	TCOM_STATE.TCOM_STATE_OP:
		// Check mapping of state:
		_bIsStateMapped := (F_GetMappingStatus(ADR(nRawState), SIZEOF(nRawState)) <> EPlcMappingStatus.MS_Unmapped);
		// Check mapping of overridden IO:
		_bIsOverriddenMapped := (F_GetMappingStatus(ADR(bRawOverridden), SIZEOF(bRawOverridden)) <> EPlcMappingStatus.MS_Unmapped);

END_CASE
END_METHOD

END_FUNCTION_BLOCK

// POUs/Local/Objects/5P/FB_BACnet_AO_Raw5P
// Analog Output Object
// - Raw communication
// - 5 Priorities
FUNCTION_BLOCK FB_BACnet_AO_Raw5P EXTENDS FB_BACnet_AO_Raw
VAR_INPUT
	bEnSfty					: BOOL;
	fValSfty				: REAL;
	bEnCrit					: BOOL;
	fValCrit				: REAL;
	bEnManLoc				: BOOL;
	fValManLoc				: REAL;
END_VAR
VAR_INPUT CONSTANT PERSISTENT
	{region 'Operational Parameters'}
		{attribute 'parameterCategory':='Manual'}
		bEnManualRm : BOOL;
		{attribute 'parameterCategory':='Manual'}
		fValManualRm : REAL;
	{endregion}
END_VAR
VAR_OUTPUT
	nActivePrio				: UDINT;			// Indicates the currently active priority of the priority array
END_VAR

SUPER^();

METHOD PROTECTED OnObjectStateChanged
SUPER^.OnObjectStateChanged();

CASE (tState) OF
	TCOM_STATE.TCOM_STATE_PREOP:
		// SyncHandler:
		RequestSyncHandlers(1, 4);
		
	TCOM_STATE.TCOM_STATE_SAFEOP:
		SyncProperty(E_BACnetPropIdentifier.PropCurrentlyActivePriority, SIZEOF(nActivePrio), ADR(nActivePrio), 0, eSync_FromSupplement, TRUE);

		SyncPropertyPvPrio(E_BACnetPropIdentifier.PropPresentValue, SIZEOF(fValSfty), ADR(fValSfty), ADR(bEnSfty), BACnet_Param.nPrio_LifeSafety, 0, eFullSync_InitPLC, TRUE);
		SyncPropertyPvPrio(E_BACnetPropIdentifier.PropPresentValue, SIZEOF(fValCrit), ADR(fValCrit), ADR(bEnCrit), BACnet_Param.nPrio_Critical, 0, eFullSync_InitPLC, TRUE);
		SyncPropertyPvPrio(E_BACnetPropIdentifier.PropPresentValue, SIZEOF(fValManLoc), ADR(fValManLoc), ADR(bEnManLoc), BACnet_Param.nPrio_ManLocal, 0, eFullSync_InitPLC, TRUE);
		SyncPropertyPvPrio(E_BACnetPropIdentifier.PropPresentValue, SIZEOF(fValManualRm), ADR(fValManualRm), ADR(bEnManualRm), BACnet_Param.nPrio_ManRemote, 0, eFullSync_InitPLC, TRUE);
		
	TCOM_STATE.TCOM_STATE_OP:
		;
		
END_CASE
END_METHOD

PROPERTY ActivePrio : UDINT
GET
ActivePrio := nActivePrio;
END_GET
END_PROPERTY

PROPERTY EnManualRm : BOOL
GET
EnManualRm := bEnManualRm;
END_GET
SET
bEnManualRm := EnManualRm;
END_SET
END_PROPERTY

PROPERTY ValManualRm : REAL
GET
ValManualRm := fValManualRm;
END_GET
SET
fValManualRm := ValManualRm;
END_SET
END_PROPERTY

END_FUNCTION_BLOCK

// POUs/Local/Objects/FB_BACnet_AO_Raw
// Analog Output Object
// - Raw communication
// - 1 Priority
FUNCTION_BLOCK FB_BACnet_AO_Raw EXTENDS FB_BACnet_BaseAO
VAR_INPUT
	bRawOverridden				: BOOL;				// Raw overridden
END_VAR
VAR_OUTPUT
	nRawValue					: INT;				// Raw value
END_VAR

IF (bReady) THEN
	// Overridden IO:
	_bOverriddenValue := bRawOverridden;
END_IF

SUPER^();

METHOD PROTECTED OnObjectStateChanged
SUPER^.OnObjectStateChanged();

CASE (tState) OF
	TCOM_STATE.TCOM_STATE_PREOP:
		// SyncHandler:
		RequestSyncHandlers(1, 0);

	TCOM_STATE.TCOM_STATE_SAFEOP:
		SyncProperty(E_BACnetPropIdentifier.PropRawIoAnalogValueINT, SIZEOF(nRawValue), ADR(nRawValue), 0, eSync_FromSupplement, TRUE);
		
	TCOM_STATE.TCOM_STATE_OP:
		;

END_CASE
END_METHOD

END_FUNCTION_BLOCK

// POUs/Local/Objects/5P/FB_BACnet_AV_5P
// Analog Value Object
// - 5 Priorities
FUNCTION_BLOCK FB_BACnet_AV_5P EXTENDS FB_BACnet_AV
VAR_INPUT
	bEnSfty					: BOOL;
	fValSfty				: REAL;
	bEnCrit					: BOOL;
	fValCrit				: REAL;
	bEnManLoc				: BOOL;
	fValManLoc				: REAL;
END_VAR
VAR_INPUT CONSTANT PERSISTENT
	{region 'Operational Parameters'}
		{attribute 'parameterCategory':='Manual'}
		bEnManualRm : BOOL;
		{attribute 'parameterCategory':='Manual'}
		fValManualRm : REAL;
	{endregion}
END_VAR
VAR_OUTPUT
	nActivePrio				: UDINT;			// Indicates the currently active priority of the priority array
END_VAR

SUPER^();

METHOD PROTECTED OnObjectStateChanged
SUPER^.OnObjectStateChanged();

CASE (tState) OF
	TCOM_STATE.TCOM_STATE_PREOP:
		// SyncHandler:
		RequestSyncHandlers(1, 4);
		
	TCOM_STATE.TCOM_STATE_SAFEOP:
		SyncProperty(E_BACnetPropIdentifier.PropCurrentlyActivePriority, SIZEOF(nActivePrio), ADR(nActivePrio), 0, eSync_FromSupplement, TRUE);

		SyncPropertyPvPrio(E_BACnetPropIdentifier.PropPresentValue, SIZEOF(fValSfty), ADR(fValSfty), ADR(bEnSfty), BACnet_Param.nPrio_LifeSafety, 0, eFullSync_InitPLC, TRUE);
		SyncPropertyPvPrio(E_BACnetPropIdentifier.PropPresentValue, SIZEOF(fValCrit), ADR(fValCrit), ADR(bEnCrit), BACnet_Param.nPrio_Critical, 0, eFullSync_InitPLC, TRUE);
		SyncPropertyPvPrio(E_BACnetPropIdentifier.PropPresentValue, SIZEOF(fValManLoc), ADR(fValManLoc), ADR(bEnManLoc), BACnet_Param.nPrio_ManLocal, 0, eFullSync_InitPLC, TRUE);
		SyncPropertyPvPrio(E_BACnetPropIdentifier.PropPresentValue, SIZEOF(fValManualRm), ADR(fValManualRm), ADR(bEnManualRm), BACnet_Param.nPrio_ManRemote, 0, eFullSync_InitPLC, TRUE);
		
	TCOM_STATE.TCOM_STATE_OP:
		;
	
END_CASE
END_METHOD

PROPERTY ActivePrio : UDINT
GET
ActivePrio := nActivePrio;
END_GET
END_PROPERTY

PROPERTY EnManualRm : BOOL
GET
EnManualRm := bEnManualRm;
END_GET
SET
bEnManualRm := EnManualRm;
END_SET
END_PROPERTY

PROPERTY ValManualRm : REAL
GET
ValManualRm := fValManualRm;
END_GET
SET
fValManualRm := ValManualRm;
END_SET
END_PROPERTY

END_FUNCTION_BLOCK

// POUs/Local/Objects/FB_BACnet_AV
// Analog Value Object
// - 1 Priority
FUNCTION_BLOCK FB_BACnet_AV EXTENDS FB_BACnet_EventObject
VAR_INPUT
	bEnPgm			: BOOL;
	fValPgm			: REAL;
END_VAR
VAR_INPUT CONSTANT PERSISTENT
	{region 'Variable Parameters'}
		{attribute 'parameterCategory':='Value'}
		fRelinquishDefault : REAL;
		{attribute 'parameterCategory':='Value'}
		bEnOutOfService : BOOL;
		{attribute 'parameterCategory':='Value'}
		fCOVIncrement : REAL := 0.1;
		{attribute 'parameterCategory':='Value'}
		eUnit : E_BA_Unit := E_BA_Unit.eOther_NoUnits;
		
		{attribute 'parameterCategory':='EventConfig'}
		bLowLimitEnable : BOOL := FALSE;
		{attribute 'parameterCategory':='EventConfig'}
		fLowLimitValue : REAL;
		{attribute 'parameterCategory':='EventConfig'}
		bHighLimitEnable : BOOL := FALSE;
		{attribute 'parameterCategory':='EventConfig'}
		fHighLimitValue : REAL;
		{attribute 'parameterCategory':='EventConfig'}
		fDeadband : REAL := 0.0;
	{endregion}
END_VAR
VAR_OUTPUT
	fPresentValue	: REAL;
END_VAR

SUPER^();

METHOD PROTECTED OnObjectStateChanged
SUPER^.OnObjectStateChanged();

CASE (tState) OF
	TCOM_STATE.TCOM_STATE_PREOP:
		// SyncHandler:
		RequestSyncHandlers(0, 9);
		
		// DisableProperty(E_BACnetPropIdentifier.PropDeviceType);

	TCOM_STATE.TCOM_STATE_SAFEOP:
		SyncPropertyPvPrio(E_BACnetPropIdentifier.PropPresentValue, SIZEOF(fValPgm), ADR(fValPgm), ADR(bEnPgm), BACnet_Param.nPrio_Program, 0, eFullSync_InitPLC, TRUE);
		
		SyncProperty(E_BACnetPropIdentifier.PropPresentValue, SIZEOF(fPresentValue), ADR(fPresentValue), 0, eSync_FromSupplement, TRUE);
		
	TCOM_STATE.TCOM_STATE_OP:
		SyncProperty(E_BACnetPropIdentifier.PropUnits, SIZEOF(eUnit), ADR(eUnit), 0, eFullSync_InitPLC, FALSE);
		SyncPropertyIdx(E_BACnetPropIdentifier.PropLimitEnable, SIZEOF(BOOL), ADR(bHighLimitEnable), E_BACnet_LimitEnableBits.eHighLimit, 0, eFullSync_InitPLC, FALSE);	
		SyncPropertyIdx(E_BACnetPropIdentifier.PropLimitEnable, SIZEOF(BOOL), ADR(bLowLimitEnable), E_BACnet_LimitEnableBits.eLowLimit, 0, eFullSync_InitPLC, FALSE);
		SyncProperty(E_BACnetPropIdentifier.PropHighLimit, SIZEOF(fHighLimitValue), ADR(fHighLimitValue), 0, eFullSync_InitPLC, FALSE);
		SyncProperty(E_BACnetPropIdentifier.PropLowLimit, SIZEOF(fLowLimitValue), ADR(fLowLimitValue), 0, eFullSync_InitPLC, FALSE);
		SyncProperty(E_BACnetPropIdentifier.PropDeadband, SIZEOF(fDeadband), ADR(fDeadband), 0, eFullSync_InitPLC, FALSE);
		SyncProperty(E_BACnetPropIdentifier.PropRelinquishDefault, SIZEOF(fRelinquishDefault), ADR(fRelinquishDefault), 0, eFullSync_InitPLC, FALSE);
		SyncProperty(E_BACnetPropIdentifier.PropOutOfService, SIZEOF(bEnOutOfService), ADR(bEnOutOfService), 0, eFullSync_InitPLC, FALSE);
		SyncProperty(E_BACnetPropIdentifier.PropCovIncrement, SIZEOF(fCOVIncrement), ADR(fCOVIncrement), 0, eFullSync_InitPLC, FALSE);
END_CASE
END_METHOD

METHOD FB_init : BOOL
VAR_INPUT
	bInitRetains : BOOL; // if TRUE, the retain variables are initialized (warm start / cold start)
	bInCopyCode : BOOL;  // if TRUE, the instance afterwards gets moved into the copy code (online change)
END_VAR
eObjectType := E_BACnetObjType.ObjAnalogValue;
END_METHOD

END_FUNCTION_BLOCK

// POUs/Local/Objects/5P/FB_BACnet_BO_IO5P
// Binary Output Object
// - Terminal communication
// - 5 Priorities
FUNCTION_BLOCK FB_BACnet_BO_IO5P EXTENDS FB_BACnet_BO_IO
VAR_INPUT
	bEnSfty					: BOOL;
	bValSfty				: BOOL;
	bEnCrit					: BOOL;
	bValCrit				: BOOL;
	bEnManLoc				: BOOL;
	bValManLoc				: BOOL;
END_VAR
VAR_INPUT CONSTANT PERSISTENT
	{region 'Operational Parameters'}
		{attribute 'parameterCategory':='Manual'}
		bEnManualRm : BOOL;
		{attribute 'parameterCategory':='Manual'}
		bValManualRm : BOOL;
	{endregion}
END_VAR
VAR_OUTPUT
	nActivePrio				: UDINT;			// Indicates the currently active priority of the priority array
END_VAR

SUPER^();

METHOD PROTECTED OnObjectStateChanged
SUPER^.OnObjectStateChanged();

CASE (tState) OF
	TCOM_STATE.TCOM_STATE_PREOP:
		// SyncHandler:
		RequestSyncHandlers(1, 4);
		
	TCOM_STATE.TCOM_STATE_SAFEOP:
		SyncProperty(E_BACnetPropIdentifier.PropCurrentlyActivePriority, SIZEOF(nActivePrio), ADR(nActivePrio), 0, eSync_FromSupplement, TRUE);

		SyncPropertyPvPrio(E_BACnetPropIdentifier.PropPresentValue, SIZEOF(bValSfty), ADR(bValSfty), ADR(bEnSfty), BACnet_Param.nPrio_LifeSafety, 0, eFullSync_InitPLC, TRUE);
		SyncPropertyPvPrio(E_BACnetPropIdentifier.PropPresentValue, SIZEOF(bValCrit), ADR(bValCrit), ADR(bEnCrit), BACnet_Param.nPrio_Critical, 0, eFullSync_InitPLC, TRUE);
		SyncPropertyPvPrio(E_BACnetPropIdentifier.PropPresentValue, SIZEOF(bValManLoc), ADR(bValManLoc), ADR(bEnManLoc), BACnet_Param.nPrio_ManLocal, 0, eFullSync_InitPLC, TRUE);
		SyncPropertyPvPrio(E_BACnetPropIdentifier.PropPresentValue, SIZEOF(bValManualRm), ADR(bValManualRm), ADR(bEnManualRm), BACnet_Param.nPrio_ManRemote, 0, eFullSync_InitPLC, TRUE);
		
	TCOM_STATE.TCOM_STATE_OP:
		;
		
END_CASE
END_METHOD

PROPERTY ActivePrio : UDINT
GET
ActivePrio := nActivePrio;
END_GET
END_PROPERTY

PROPERTY EnManualRm : BOOL
GET
EnManualRm := bEnManualRm;
END_GET
SET
bEnManualRm := EnManualRm;
END_SET
END_PROPERTY

PROPERTY ValManualRm : BOOL
GET
ValManualRm := bValManualRm;
END_GET
SET
bValManualRm := ValManualRm;
END_SET
END_PROPERTY

END_FUNCTION_BLOCK

// POUs/Local/Objects/FB_BACnet_BO_IO
// Binary Output Object
// - Terminal communication
// - 1 Priority
FUNCTION_BLOCK FB_BACnet_BO_IO EXTENDS FB_BACnet_BaseBO
VAR_INPUT CONSTANT PERSISTENT
	{region 'Variable Parameters'}
		{attribute 'parameterCategory':='Config'}
		eFeedbackPolarity : E_BA_Polarity := E_BA_Polarity.eNormal;
		{attribute 'parameterCategory':='Config'}
		eOverriddenPolarity : E_BA_Polarity := E_BA_Polarity.eNormal;
	{endregion}
END_VAR
VAR
	{region 'Raw I/O'}
		bRawOverridden		AT %I*	: BOOL;				// Raw overridden (Optional)
		bRawValFeedback		AT %I*	: BOOL;				// Raw feedback Value (Optional)
		bRawValue			AT %Q*	: BOOL;				// Raw value
	{endregion}
	{region 'Hardware'}
		_bIsFeedbackMapped			: BOOL;				// Indication to mapped hardware for feedback value
		_bIsOverriddenMapped		: BOOL;				// Indication to mapped hardware for overridden IO value
	{endregion}
	{region 'Internal'}
		_bOverriddenValue			: BOOL;
	{endregion}
END_VAR
VAR_STAT 
	// (BETA) ... Following symbols should be made non-static / thread safe!
	{region 'Temporary'}
		{attribute 'hide'}
		_bEnFeedback				: BOOL;
	{endregion}
END_VAR

IF (bReady) THEN
	// Overridden IO Value:
	_bOverriddenValue := SEL(_bIsOverriddenMapped, FALSE, (bRawOverridden = (eOverriddenPolarity=E_BA_Polarity.eNormal)));
	
	// Feedback Value:
	_bEnFeedback := SEL(_bIsFeedbackMapped, FALSE, NOT _bOverriddenValue);
	_bFeedbackValue := SEL(_bEnFeedback, bPresentValue, (bRawValFeedback = (eFeedbackPolarity=E_BA_Polarity.eNormal)));
END_IF

SUPER^();

METHOD PROTECTED OnObjectStateChanged
SUPER^.OnObjectStateChanged();

CASE (tState) OF
	TCOM_STATE.TCOM_STATE_PREOP:
		// SyncHandler:
		RequestSyncHandlers(1, 1);

	TCOM_STATE.TCOM_STATE_SAFEOP:
		SyncProperty(E_BACnetPropIdentifier.PropRawIoBinaryValueBOOL, SIZEOF(bRawValue), ADR(bRawValue), 0, eSync_FromSupplement, TRUE);
		
	TCOM_STATE.TCOM_STATE_OP:
		SyncProperty(E_BACnetPropIdentifier.PropRawIoStateOverrideInverted, SIZEOF(_bOverriddenValue), ADR(_bOverriddenValue), 0, eSync_ToSupplement, FALSE);

		// Check mapping of feedback:
		_bIsFeedbackMapped := (F_GetMappingStatus(ADR(bRawValFeedback), SIZEOF(bRawValFeedback)) <> EPlcMappingStatus.MS_Unmapped);
		// Check mapping of overridden IO:
		_bIsOverriddenMapped := (F_GetMappingStatus(ADR(bRawOverridden), SIZEOF(bRawOverridden)) <> EPlcMappingStatus.MS_Unmapped);
		
END_CASE
END_METHOD

END_FUNCTION_BLOCK

// POUs/Local/Objects/5P/FB_BACnet_BO_Raw5P
// Binary Output Object
// - Raw communication
// - 5 Priorities
FUNCTION_BLOCK FB_BACnet_BO_Raw5P EXTENDS FB_BACnet_BO_Raw
VAR_INPUT
	bEnSfty					: BOOL;
	bValSfty				: BOOL;
	bEnCrit					: BOOL;
	bValCrit				: BOOL;
	bEnManLoc				: BOOL;
	bValManLoc				: BOOL;
END_VAR
VAR_INPUT CONSTANT PERSISTENT
	{region 'Operational Parameters'}
		{attribute 'parameterCategory':='Manual'}
		bEnManualRm : BOOL;
		{attribute 'parameterCategory':='Manual'}
		bValManualRm : BOOL;
	{endregion}
END_VAR
VAR_OUTPUT
	nActivePrio				: UDINT;			// Indicates the currently active priority of the priority array
END_VAR

SUPER^();

METHOD PROTECTED OnObjectStateChanged
SUPER^.OnObjectStateChanged();

CASE (tState) OF
	TCOM_STATE.TCOM_STATE_PREOP:
		// SyncHandler:
		RequestSyncHandlers(1, 4);
		
	TCOM_STATE.TCOM_STATE_SAFEOP:
		SyncProperty(E_BACnetPropIdentifier.PropCurrentlyActivePriority, SIZEOF(nActivePrio), ADR(nActivePrio), 0, eSync_FromSupplement, TRUE);

		SyncPropertyPvPrio(E_BACnetPropIdentifier.PropPresentValue, SIZEOF(bValSfty), ADR(bValSfty), ADR(bEnSfty), BACnet_Param.nPrio_LifeSafety, 0, eFullSync_InitPLC, TRUE);
		SyncPropertyPvPrio(E_BACnetPropIdentifier.PropPresentValue, SIZEOF(bValCrit), ADR(bValCrit), ADR(bEnCrit), BACnet_Param.nPrio_Critical, 0, eFullSync_InitPLC, TRUE);
		SyncPropertyPvPrio(E_BACnetPropIdentifier.PropPresentValue, SIZEOF(bValManLoc), ADR(bValManLoc), ADR(bEnManLoc), BACnet_Param.nPrio_ManLocal, 0, eFullSync_InitPLC, TRUE);
		SyncPropertyPvPrio(E_BACnetPropIdentifier.PropPresentValue, SIZEOF(bValManualRm), ADR(bValManualRm), ADR(bEnManualRm), BACnet_Param.nPrio_ManRemote, 0, eFullSync_InitPLC, TRUE);
		
	TCOM_STATE.TCOM_STATE_OP:
		;
		
END_CASE
END_METHOD

PROPERTY ActivePrio : UDINT
GET
ActivePrio := nActivePrio;
END_GET
END_PROPERTY

PROPERTY EnManualRm : BOOL
GET
EnManualRm := bEnManualRm;
END_GET
SET
bEnManualRm := EnManualRm;
END_SET
END_PROPERTY

PROPERTY ValManualRm : BOOL
GET
ValManualRm := bValManualRm;
END_GET
SET
bValManualRm := ValManualRm;
END_SET
END_PROPERTY

END_FUNCTION_BLOCK

// POUs/Local/Objects/FB_BACnet_BO_Raw
// Binary Output Object
// - Raw communication
// - 1 Priority
FUNCTION_BLOCK FB_BACnet_BO_Raw EXTENDS FB_BACnet_BaseBO
VAR_INPUT
	bRawOverridden				: BOOL;				// Raw overridden

	bEnFeedback					: BOOL;				// Enable of writing to Feedback Value (optional)
	bRawValFeedback				: BOOL;				// Raw feedback Value
END_VAR
VAR_OUTPUT
	bRawValue					: BOOL;				// Raw value
END_VAR

IF (bReady) THEN
	// Feedback Value:
	_bFeedbackValue := SEL(bEnFeedback, bPresentValue, bRawValFeedback);
END_IF

SUPER^();

METHOD PROTECTED OnObjectStateChanged
SUPER^.OnObjectStateChanged();

CASE (tState) OF
	TCOM_STATE.TCOM_STATE_PREOP:
		// SyncHandler:
		RequestSyncHandlers(1, 1);

	TCOM_STATE.TCOM_STATE_SAFEOP:
		SyncProperty(E_BACnetPropIdentifier.PropRawIoBinaryValueBOOL, SIZEOF(bRawValue), ADR(bRawValue), 0, eSync_FromSupplement, TRUE);
		
	TCOM_STATE.TCOM_STATE_OP:
		SyncProperty(E_BACnetPropIdentifier.PropRawIoStateOverrideInverted, SIZEOF(bRawOverridden), ADR(bRawOverridden), 0, eSync_ToSupplement, FALSE);

END_CASE
END_METHOD

END_FUNCTION_BLOCK

// POUs/Local/Objects/5P/FB_BACnet_BV_5P
// Binary Value Object
// - 5 Priorities
FUNCTION_BLOCK FB_BACnet_BV_5P EXTENDS FB_BACnet_BV
VAR_INPUT
	bEnSfty					: BOOL;
	bValSfty				: BOOL;
	bEnCrit					: BOOL;
	bValCrit				: BOOL;
	bEnManLoc				: BOOL;
	bValManLoc				: BOOL;
END_VAR
VAR_INPUT CONSTANT PERSISTENT
	{region 'Operational Parameters'}
		{attribute 'parameterCategory':='Manual'}
		bEnManualRm : BOOL;
		{attribute 'parameterCategory':='Manual'}
		bValManualRm : BOOL;
	{endregion}
END_VAR
VAR_OUTPUT
	nActivePrio				: UDINT;			// Indicates the currently active priority of the priority array
END_VAR

SUPER^();

METHOD PROTECTED OnObjectStateChanged
SUPER^.OnObjectStateChanged();

CASE (tState) OF
	TCOM_STATE.TCOM_STATE_PREOP:
		// SyncHandler:
		RequestSyncHandlers(1, 4);
		
	TCOM_STATE.TCOM_STATE_SAFEOP:
		SyncProperty(E_BACnetPropIdentifier.PropCurrentlyActivePriority, SIZEOF(nActivePrio), ADR(nActivePrio), 0, eSync_FromSupplement, TRUE);

		SyncPropertyPvPrio(E_BACnetPropIdentifier.PropPresentValue, SIZEOF(bValSfty), ADR(bValSfty), ADR(bEnSfty), BACnet_Param.nPrio_LifeSafety, 0, eFullSync_InitPLC, TRUE);
		SyncPropertyPvPrio(E_BACnetPropIdentifier.PropPresentValue, SIZEOF(bValCrit), ADR(bValCrit), ADR(bEnCrit), BACnet_Param.nPrio_Critical, 0, eFullSync_InitPLC, TRUE);
		SyncPropertyPvPrio(E_BACnetPropIdentifier.PropPresentValue, SIZEOF(bValManLoc), ADR(bValManLoc), ADR(bEnManLoc), BACnet_Param.nPrio_ManLocal, 0, eFullSync_InitPLC, TRUE);
		SyncPropertyPvPrio(E_BACnetPropIdentifier.PropPresentValue, SIZEOF(bValManualRm), ADR(bValManualRm), ADR(bEnManualRm), BACnet_Param.nPrio_ManRemote, 0, eFullSync_InitPLC, TRUE);
		
	TCOM_STATE.TCOM_STATE_OP:
		;
		
END_CASE
END_METHOD

PROPERTY ActivePrio : UDINT
GET
ActivePrio := nActivePrio;
END_GET
END_PROPERTY

PROPERTY EnManualRm : BOOL
GET
EnManualRm := bEnManualRm;
END_GET
SET
bEnManualRm := EnManualRm;
END_SET
END_PROPERTY

PROPERTY ValManualRm : BOOL
GET
ValManualRm := bValManualRm;
END_GET
SET
bValManualRm := ValManualRm;
END_SET
END_PROPERTY

END_FUNCTION_BLOCK

// POUs/Local/Objects/FB_BACnet_BV
// Binary Value Object
// - 1 Priority
FUNCTION_BLOCK FB_BACnet_BV EXTENDS FB_BACnet_EventObject
VAR_INPUT
	bEnPgm		: BOOL;
	bValPgm		: BOOL;
END_VAR
VAR_INPUT CONSTANT PERSISTENT
	{region 'Variable Parameters'}
		{attribute 'parameterCategory':='General'}
		{attribute 'parameterUnit':= 's'}
		nMinimumOffTime : UDINT;
		{attribute 'parameterCategory':='General'}
		{attribute 'parameterUnit':= 's'}
		nMinimumOnTime : UDINT;
		
		{attribute 'parameterCategory':='Value'}
		bRelinquishDefault : BOOL;
		{attribute 'parameterCategory':='Value'}
		bEnOutOfService : BOOL;
		{attribute 'parameterCategory':='Value'}
		{attribute 'TcEncoding':='UTF-8'}
		sInactiveText : T_BACnet_StateText;
		{attribute 'parameterCategory':='Value'}
		{attribute 'TcEncoding':='UTF-8'}
		sActiveText : T_BACnet_StateText;
		
		{attribute 'parameterCategory':='EventConfig'}
		bAlarmValue : BOOL := TRUE;
			 
		{attribute 'parameterCategory':='StateChange'}
		nChangeOfStateCount : UDINT;
		
		{attribute 'parameterCategory':='ActiveTime'}
		{attribute 'parameterUnit':= 's'}
		nElapsedActiveTime : UDINT;
	{endregion}
END_VAR
VAR_OUTPUT
	bPresentValue	: BOOL;
END_VAR
VAR
	{region 'Output-Properties'}
		{attribute 'parameterCategory':='StateChange'}
		stChangeOfStateTime : ST_BA_DateTime;
		{attribute 'parameterCategory':='StateChange'}
		stTimeOfStateCountReset : ST_BA_DateTime;
		
		{attribute 'parameterCategory':='ActiveTime'}
		stTimeOfActiveTimeReset : ST_BA_DateTime;
	{endregion}
END_VAR

SUPER^();

METHOD PROTECTED OnObjectStateChanged
SUPER^.OnObjectStateChanged();

CASE (tState) OF
	TCOM_STATE.TCOM_STATE_PREOP:
		// SyncHandler:
		RequestSyncHandlers(4, 10);
		
		// Properties:
		EnableProperty(E_BACnetPropIdentifier.PropDeviceType, FALSE);

		IF (BACnet_Param.bStateText_WriteProtect) THEN
			WriteProtectProperty(E_BACnetPropIdentifier.PropActiveText, TRUE);
			WriteProtectProperty(E_BACnetPropIdentifier.PropInactiveText, TRUE);
		END_IF
		
		// Ensure UTF-8 Encoding:
		F_BA_EnsureUTF8(ADR(sInactiveText), SIZEOF(sInactiveText));
		F_BA_EnsureUTF8(ADR(sActiveText), SIZEOF(sActiveText));

	TCOM_STATE.TCOM_STATE_SAFEOP:
		SyncPropertyPvPrio(E_BACnetPropIdentifier.PropPresentValue, SIZEOF(bValPgm), ADR(bValPgm), ADR(bEnPgm), BACnet_Param.nPrio_Program, 0, eFullSync_InitPLC, TRUE);
		
		SyncProperty(E_BACnetPropIdentifier.PropPresentValue, SIZEOF(bPresentValue), ADR(bPresentValue), 0, eSync_FromSupplement, TRUE);
		
	TCOM_STATE.TCOM_STATE_OP:
		SyncProperty(E_BACnetPropIdentifier.PropAlarmValue, SIZEOF(bAlarmValue), ADR(bAlarmValue), 0, eFullSync_InitPLC, FALSE);
		SyncProperty(E_BACnetPropIdentifier.PropOutOfService, SIZEOF(bEnOutOfService), ADR(bEnOutOfService), 0, eFullSync_InitPLC, FALSE);
		SyncProperty(E_BACnetPropIdentifier.PropMinimumOffTime, SIZEOF(nMinimumOffTime), ADR(nMinimumOffTime), 0, eFullSync_InitPLC, FALSE);	
		SyncProperty(E_BACnetPropIdentifier.PropMinimumOnTime, SIZEOF(nMinimumOnTime), ADR(nMinimumOnTime), 0, eFullSync_InitPLC, FALSE);	
		SyncProperty(E_BACnetPropIdentifier.PropRelinquishDefault, SIZEOF(bRelinquishDefault), ADR(bRelinquishDefault), 0, eFullSync_InitPLC, FALSE);	
		SyncProperty(E_BACnetPropIdentifier.PropActiveText, SIZEOF(sActiveText), ADR(sActiveText), 0, eFullSync_InitPLC, FALSE);	
		SyncProperty(E_BACnetPropIdentifier.PropInactiveText, SIZEOF(sInactiveText), ADR(sInactiveText), 0, eFullSync_InitPLC, FALSE);

		SyncProperty(E_BACnetPropIdentifier.PropChangeOfStateCount, SIZEOF(nChangeOfStateCount), ADR(nChangeOfStateCount), 0, eFullSync_InitPLC, FALSE);
		SyncProperty(E_BACnetPropIdentifier.PropChangeOfStateTime, SIZEOF(stChangeOfStateTime), ADR(stChangeOfStateTime), 0, eSync_FromSupplement, FALSE);
		SyncProperty(E_BACnetPropIdentifier.PropTimeOfStateCountReset, SIZEOF(stTimeOfStateCountReset), ADR(stTimeOfStateCountReset), 0, eSync_FromSupplement, FALSE);

		SyncProperty(E_BACnetPropIdentifier.PropElapsedActiveTime, SIZEOF(nElapsedActiveTime), ADR(nElapsedActiveTime), 0, eFullSync_InitPLC, FALSE);
		SyncProperty(E_BACnetPropIdentifier.PropTimeOfActiveTimeReset, SIZEOF(stTimeOfActiveTimeReset), ADR(stTimeOfActiveTimeReset), 0, eSync_FromSupplement, FALSE);
		
END_CASE
END_METHOD

METHOD FB_init : BOOL
VAR_INPUT
	bInitRetains : BOOL; // if TRUE, the retain variables are initialized (warm start / cold start)
	bInCopyCode : BOOL;  // if TRUE, the instance afterwards gets moved into the copy code (online change)
END_VAR
eObjectType := E_BACnetObjType.ObjBinaryValue;
END_METHOD

END_FUNCTION_BLOCK

// POUs/Local/Objects/5P/FB_BACnet_MO_IO5P
// Multistate Output Object
// - Terminal communication
// - 5 Priorities
FUNCTION_BLOCK FB_BACnet_MO_IO5P EXTENDS FB_BACnet_MO_IO
VAR_INPUT
	bEnSfty					: BOOL;
	nValSfty				: UDINT		:= 1;
	bEnCrit					: BOOL;
	nValCrit				: UDINT		:= 1;
	bEnManLoc				: BOOL;
	nValManLoc				: UDINT		:= 1;
END_VAR
VAR_INPUT CONSTANT PERSISTENT
	{region 'Operational Parameters'}
		{attribute 'parameterCategory':='Manual'}
		bEnManualRm : BOOL;
		{attribute 'parameterCategory':='Manual'}
		nValManualRm : UDINT := 1;
	{endregion}
END_VAR
VAR_OUTPUT
	nActivePrio				: UDINT;					// Indicates the currently active priority of the priority array
END_VAR

SUPER^();

METHOD PROTECTED OnObjectStateChanged
SUPER^.OnObjectStateChanged();

CASE (tState) OF
	TCOM_STATE.TCOM_STATE_PREOP:
		// SyncHandler:
		RequestSyncHandlers(1, 4);
		
	TCOM_STATE.TCOM_STATE_SAFEOP:
		SyncProperty(E_BACnetPropIdentifier.PropCurrentlyActivePriority, SIZEOF(nActivePrio), ADR(nActivePrio), 0, eSync_FromSupplement, TRUE);

		SyncPropertyPvPrio(E_BACnetPropIdentifier.PropPresentValue, SIZEOF(nValSfty), ADR(nValSfty), ADR(bEnSfty), BACnet_Param.nPrio_LifeSafety, 0, eFullSync_InitPLC, TRUE);
		SyncPropertyPvPrio(E_BACnetPropIdentifier.PropPresentValue, SIZEOF(nValCrit), ADR(nValCrit), ADR(bEnCrit), BACnet_Param.nPrio_Critical, 0, eFullSync_InitPLC, TRUE);
		SyncPropertyPvPrio(E_BACnetPropIdentifier.PropPresentValue, SIZEOF(nValManLoc), ADR(nValManLoc), ADR(bEnManLoc), BACnet_Param.nPrio_ManLocal, 0, eFullSync_InitPLC, TRUE);
		SyncPropertyPvPrio(E_BACnetPropIdentifier.PropPresentValue, SIZEOF(nValManualRm), ADR(nValManualRm), ADR(bEnManualRm), BACnet_Param.nPrio_ManRemote, 0, eFullSync_InitPLC, TRUE);
		
	TCOM_STATE.TCOM_STATE_OP:
		;
		
END_CASE
END_METHOD

PROPERTY ActivePrio : UDINT
GET
ActivePrio := nActivePrio;
END_GET
END_PROPERTY

PROPERTY EnManualRm : BOOL
GET
EnManualRm := bEnManualRm;
END_GET
SET
bEnManualRm := EnManualRm;
END_SET
END_PROPERTY

PROPERTY ValManualRm : UDINT
GET
ValManualRm := nValManualRm;
END_GET
SET
nValManualRm := ValManualRm;
END_SET
END_PROPERTY

END_FUNCTION_BLOCK

// POUs/Local/Objects/FB_BACnet_MO_IO
// Multistate Output Object
// - Terminal communication
// - 1 Priority
FUNCTION_BLOCK FB_BACnet_MO_IO EXTENDS FB_BACnet_BaseMO
VAR_INPUT CONSTANT PERSISTENT
	{region 'Variable Parameters'}
		{attribute 'parameterCategory':='Config'}
		eMappingMode : E_BA_ByteMappingMode := E_BA_ByteMappingMode.eIndex1N;
		{attribute 'parameterCategory':='Config'}
		eFeedbackMappingMode : E_BA_ByteMappingMode := E_BA_ByteMappingMode.eIndex1N;
	{endregion}
END_VAR
VAR
	{region 'Raw I/O'}
		bRawValFeedback		AT %I*	: ST_BA_Byte;		// Bus terminal feedback Value (Optional)
		bRawValue			AT %Q*	: ST_BA_Byte;		// Bus terminal value
	{endregion}
	{region 'Hardware'}
		_bIsFeedbackMapped			: BOOL;				// Indication to mapped hardware for feedback value
	{endregion}
	{region 'Internal'}
		nLastPresentValue			: UDINT;
	{endregion}
END_VAR

IF (bReady) THEN
	// Feedback Value:
	IF (_bIsFeedbackMapped) THEN
		F_BA_MapUDIFromRawByte(bRawValFeedback, _nFeedbackValue, eFeedbackMappingMode, nRelinquishDefault);
	ELSE
		_nFeedbackValue := nPresentValue;
	END_IF
	
	// Trigger change of value:
	IF (nPresentValue <> nLastPresentValue) THEN
		nLastPresentValue := nPresentValue;
		F_BA_MapUDIToRawByte(bRawValue, nPresentValue, eMappingMode, nRelinquishDefault);
	END_IF
ELSE
	nPresentValue := nRelinquishDefault;
	
	// Set last value to a different value compared to actual raw value (So a COV is triggered when current instance becomes ready):
	nLastPresentValue := (nLastPresentValue+1);
END_IF

SUPER^();

METHOD PROTECTED OnObjectStateChanged
SUPER^.OnObjectStateChanged();

CASE (tState) OF
	TCOM_STATE.TCOM_STATE_PREOP:
		;

	TCOM_STATE.TCOM_STATE_SAFEOP:
		;
		
	TCOM_STATE.TCOM_STATE_OP:
		// Check mapping of feedback:
		_bIsFeedbackMapped := (F_GetMappingStatus(ADR(bRawValFeedback), SIZEOF(bRawValFeedback)) <> EPlcMappingStatus.MS_Unmapped);
		
END_CASE
END_METHOD

END_FUNCTION_BLOCK

// POUs/Local/Objects/5P/FB_BACnet_MO_Raw5P
// Multistate Output Object
// - Raw communication
// - 5 Priorities
FUNCTION_BLOCK FB_BACnet_MO_Raw5P EXTENDS FB_BACnet_MO_Raw
VAR_INPUT
	bEnSfty					: BOOL;
	nValSfty				: UDINT		:= 1;
	bEnCrit					: BOOL;
	nValCrit				: UDINT		:= 1;
	bEnManLoc				: BOOL;
	nValManLoc				: UDINT		:= 1;
END_VAR
VAR_INPUT CONSTANT PERSISTENT
	{region 'Operational Parameters'}
		{attribute 'parameterCategory':='Manual'}
		bEnManualRm : BOOL;
		{attribute 'parameterCategory':='Manual'}
		nValManualRm : UDINT := 1;
	{endregion}
END_VAR
VAR_OUTPUT
	nActivePrio				: UDINT;					// Indicates the currently active priority of the priority array
END_VAR

SUPER^();

METHOD PROTECTED OnObjectStateChanged
SUPER^.OnObjectStateChanged();

CASE (tState) OF
	TCOM_STATE.TCOM_STATE_PREOP:
		// SyncHandler:
		RequestSyncHandlers(1, 4);
		
	TCOM_STATE.TCOM_STATE_SAFEOP:
		SyncProperty(E_BACnetPropIdentifier.PropCurrentlyActivePriority, SIZEOF(nActivePrio), ADR(nActivePrio), 0, eSync_FromSupplement, TRUE);

		SyncPropertyPvPrio(E_BACnetPropIdentifier.PropPresentValue, SIZEOF(nValSfty), ADR(nValSfty), ADR(bEnSfty), BACnet_Param.nPrio_LifeSafety, 0, eFullSync_InitPLC, TRUE);
		SyncPropertyPvPrio(E_BACnetPropIdentifier.PropPresentValue, SIZEOF(nValCrit), ADR(nValCrit), ADR(bEnCrit), BACnet_Param.nPrio_Critical, 0, eFullSync_InitPLC, TRUE);
		SyncPropertyPvPrio(E_BACnetPropIdentifier.PropPresentValue, SIZEOF(nValManLoc), ADR(nValManLoc), ADR(bEnManLoc), BACnet_Param.nPrio_ManLocal, 0, eFullSync_InitPLC, TRUE);
		SyncPropertyPvPrio(E_BACnetPropIdentifier.PropPresentValue, SIZEOF(nValManualRm), ADR(nValManualRm), ADR(bEnManualRm), BACnet_Param.nPrio_ManRemote, 0, eFullSync_InitPLC, TRUE);
		
	TCOM_STATE.TCOM_STATE_OP:
		;
		
END_CASE
END_METHOD

PROPERTY ActivePrio : UDINT
GET
ActivePrio := nActivePrio;
END_GET
END_PROPERTY

PROPERTY EnManualRm : BOOL
GET
EnManualRm := bEnManualRm;
END_GET
SET
bEnManualRm := EnManualRm;
END_SET
END_PROPERTY

PROPERTY ValManualRm : UDINT
GET
ValManualRm := nValManualRm;
END_GET
SET
nValManualRm := ValManualRm;
END_SET
END_PROPERTY

END_FUNCTION_BLOCK

// POUs/Local/Objects/FB_BACnet_MO_Raw
// Multistate Output Object
// - Raw communication
// - 1 Priority
FUNCTION_BLOCK FB_BACnet_MO_Raw EXTENDS FB_BACnet_BaseMO
VAR_INPUT
	bEnFeedback					: BOOL;				// Enable of writing to Feedback Value (optional)
	nRawValFeedback				: UDINT;			// Raw feedback Value
END_VAR
VAR_OUTPUT
	nRawValue					: UDINT;			// Raw value
END_VAR

IF (bReady) THEN
	// Feedback Value:
	_nFeedbackValue := MAX(1, SEL(bEnFeedback, nPresentValue, nRawValFeedback));
	
	// Raw-IO Value:
	nRawValue := nPresentValue;
END_IF

SUPER^();

END_FUNCTION_BLOCK

// POUs/Local/Objects/5P/FB_BACnet_MV_5P
// Multistate Value Object
// - 5 Priorities
FUNCTION_BLOCK FB_BACnet_MV_5P EXTENDS FB_BACnet_MV
VAR_INPUT
	bEnSfty					: BOOL;
	nValSfty				: UDINT		:= 1;
	bEnCrit					: BOOL;
	nValCrit				: UDINT		:= 1;
	bEnManLoc				: BOOL;
	nValManLoc				: UDINT		:= 1;
END_VAR
VAR_INPUT CONSTANT PERSISTENT
	{region 'Operational Parameters'}
		{attribute 'parameterCategory':='Manual'}
		bEnManualRm : BOOL;
		{attribute 'parameterCategory':='Manual'}
		nValManualRm : UDINT := 1;
	{endregion}
END_VAR
VAR_OUTPUT
	nActivePrio				: UDINT;			// Indicates the currently active priority of the priority array
END_VAR

SUPER^();

METHOD PROTECTED OnObjectStateChanged
SUPER^.OnObjectStateChanged();

CASE (tState) OF
	TCOM_STATE.TCOM_STATE_PREOP:
		// SyncHandler:
		RequestSyncHandlers(1, 4);
		
	TCOM_STATE.TCOM_STATE_SAFEOP:
		SyncProperty(E_BACnetPropIdentifier.PropCurrentlyActivePriority, SIZEOF(nActivePrio), ADR(nActivePrio), 0, eSync_FromSupplement, TRUE);

		SyncPropertyPvPrio(E_BACnetPropIdentifier.PropPresentValue, SIZEOF(nValSfty), ADR(nValSfty), ADR(bEnSfty), BACnet_Param.nPrio_LifeSafety, 0, eFullSync_InitPLC, TRUE);
		SyncPropertyPvPrio(E_BACnetPropIdentifier.PropPresentValue, SIZEOF(nValCrit), ADR(nValCrit), ADR(bEnCrit), BACnet_Param.nPrio_Critical, 0, eFullSync_InitPLC, TRUE);
		SyncPropertyPvPrio(E_BACnetPropIdentifier.PropPresentValue, SIZEOF(nValManLoc), ADR(nValManLoc), ADR(bEnManLoc), BACnet_Param.nPrio_ManLocal, 0, eFullSync_InitPLC, TRUE);
		SyncPropertyPvPrio(E_BACnetPropIdentifier.PropPresentValue, SIZEOF(nValManualRm), ADR(nValManualRm), ADR(bEnManualRm), BACnet_Param.nPrio_ManRemote, 0, eFullSync_InitPLC, TRUE);
		
	TCOM_STATE.TCOM_STATE_OP:
		;
		
END_CASE
END_METHOD

PROPERTY ActivePrio : UDINT
GET
ActivePrio := nActivePrio;
END_GET
END_PROPERTY

PROPERTY EnManualRm : BOOL
GET
EnManualRm := bEnManualRm;
END_GET
SET
bEnManualRm := EnManualRm;
END_SET
END_PROPERTY

PROPERTY ValManualRm : UDINT
GET
ValManualRm := nValManualRm;
END_GET
SET
nValManualRm := ValManualRm;
END_SET
END_PROPERTY

END_FUNCTION_BLOCK

// POUs/Local/Objects/FB_BACnet_MV
// Multistate Value Object
// - 1 Priority
FUNCTION_BLOCK FB_BACnet_MV EXTENDS FB_BACnet_EventObject
VAR_INPUT
	bEnPgm					: BOOL;
	nValPgm					: UDINT		:= 1;
END_VAR
VAR_INPUT CONSTANT PERSISTENT
	{region 'Fixed Parameters'}
		{attribute 'parameterCategory':='Value'}
		{attribute 'TcEncoding':='UTF-8'}
		sStateText : ARRAY[1..BACnet_Param.nMultistate_StateCount] OF T_BACnet_StateText;
		
		{attribute 'parameterCategory':='EventConfig'}
		nAlarmValues : ARRAY[1..BACnet_Param.nMultistate_StateCount] OF UDINT;
		{attribute 'parameterCategory':='EventConfig'}
		nFaultValues : ARRAY[1..BACnet_Param.nMultistate_StateCount] OF UDINT;
	{endregion}
	{region 'Variable Parameters'}
		{attribute 'parameterCategory':='Value'}
		nRelinquishDefault : UDINT := 1;
		{attribute 'parameterCategory':='Value'}
		bEnOutOfService : BOOL;
	{endregion}
END_VAR
VAR_OUTPUT
	nPresentValue			: UDINT		:= 1;
END_VAR
VAR
	{region 'Output-Properties'}
		nStateCount			: UDINT;
	{endregion}
END_VAR

SUPER^();

METHOD PROTECTED OnObjectStateChanged
SUPER^.OnObjectStateChanged();

CASE (tState) OF
	TCOM_STATE.TCOM_STATE_PREOP:
		// SyncHandler:
		{warning disable C0196}
		nStateCount := F_BACnet_GetUsedStateText(sStateText);
		{warning restore C0196}
		
		RequestSyncHandlers(0, nStateCount);								// Handlers for "E_BACnetPropIdentifier.PropStateText"
		RequestSyncHandlers(0, F_BACnet_GetUsedUDINT(nAlarmValues));		// Handlers for "E_BACnetPropIdentifier.PropAlarmValues"
		RequestSyncHandlers(0, F_BACnet_GetUsedUDINT(nFaultValues));		// Handlers for "E_BACnetPropIdentifier.PropFaultValues"
		RequestSyncHandlers(1, 3);											// Handlers for other properties
		
		// Properties:
		EnableProperty(E_BACnetPropIdentifier.PropDeviceType, FALSE);
		
		WriteProtectProperty(E_BACnetPropIdentifier.PropNumberOfStates, TRUE);
		
		IF (BACnet_Param.bStateText_WriteProtect) THEN
			WriteProtectProperty(E_BACnetPropIdentifier.PropStateText, TRUE);
		END_IF
		
		// Ensure UTF-8 Encoding:
		F_BA_EnsureUTF8Array(ADR(sStateText), SIZEOF(sStateText[1]), TO_DINT(BACnet_Param.nMultistate_StateCount));
		
	TCOM_STATE.TCOM_STATE_SAFEOP:
		SyncPropertyPvPrio(E_BACnetPropIdentifier.PropPresentValue, SIZEOF(nValPgm), ADR(nValPgm), ADR(bEnPgm), BACnet_Param.nPrio_Program, 0, eFullSync_InitPLC, TRUE);
		
		SyncProperty(E_BACnetPropIdentifier.PropPresentValue, SIZEOF(nPresentValue), ADR(nPresentValue), 0, eSync_FromSupplement, TRUE);
		
	TCOM_STATE.TCOM_STATE_OP:
		// Init number of used states:
		SetNumberOfStates(nStateCount);
		
		SyncProperty(E_BACnetPropIdentifier.PropRelinquishDefault, SIZEOF(nRelinquishDefault), ADR(nRelinquishDefault), 0, eFullSync_InitPLC, FALSE);
		SyncProperty(E_BACnetPropIdentifier.PropOutOfService, SIZEOF(bEnOutOfService), ADR(bEnOutOfService), 0, eFullSync_InitPLC, FALSE);
		SyncPropertyList(E_BACnetPropIdentifier.PropStateText, ADR(sStateText), SIZEOF(T_BACnet_StateText), nStateCount, eFullSync_InitPLC, FALSE);
		SyncPropertyList(E_BACnetPropIdentifier.PropAlarmValues, ADR(nAlarmValues), SIZEOF(UDINT), nStateCount, eFullSync_InitPLC, TRUE);
		SyncPropertyList(E_BACnetPropIdentifier.PropFaultValues, ADR(nFaultValues), SIZEOF(UDINT), nStateCount, eFullSync_InitPLC, TRUE);
		
END_CASE
END_METHOD

METHOD FB_init : BOOL
VAR_INPUT
	bInitRetains : BOOL; // if TRUE, the retain variables are initialized (warm start / cold start)
	bInCopyCode : BOOL;  // if TRUE, the instance afterwards gets moved into the copy code (online change)
END_VAR
eObjectType := E_BACnetObjType.ObjMultistateValue;
END_METHOD

PROPERTY StateCount : UDINT
GET
StateCount := nStateCount;
END_GET
END_PROPERTY

END_FUNCTION_BLOCK

// POUs/Local/Objects/FB_BACnet_Acc
// Accumulator Object
FUNCTION_BLOCK FB_BACnet_Acc EXTENDS FB_BACnet_EventObject
VAR_OUTPUT
	nPresentValue			: UDINT;
END_VAR

SUPER^();

METHOD PROTECTED OnObjectStateChanged
SUPER^.OnObjectStateChanged();

CASE (tState) OF
	TCOM_STATE.TCOM_STATE_PREOP:
		// SyncHandler:
		RequestSyncHandlers(1, 0);
		
	TCOM_STATE.TCOM_STATE_SAFEOP:
		SyncProperty(E_BACnetPropIdentifier.PropPresentValue, SIZEOF(nPresentValue), ADR(nPresentValue), 0, eSync_FromSupplement, TRUE);
	
	TCOM_STATE.TCOM_STATE_OP:
		;
		
END_CASE
END_METHOD

METHOD FB_init : BOOL
VAR_INPUT
	bInitRetains : BOOL; // if TRUE, the retain variables are initialized (warm start / cold start)
	bInCopyCode : BOOL;  // if TRUE, the instance afterwards gets moved into the copy code (online change)
END_VAR
eObjectType := E_BACnetObjType.ObjAccumulator;
END_METHOD

END_FUNCTION_BLOCK

// POUs/Local/Objects/FB_BACnet_AI
// Analog Input Object
// - process value
FUNCTION_BLOCK FB_BACnet_AI EXTENDS FB_BACnet_BaseAI
VAR_INPUT
	fVal						: REAL;				// Process value
END_VAR

IF bReady THEN
	IF NOT bEnOutOfService THEN
		fPresentValue := fVal;
	END_IF
ELSE
	fPresentValue := 0;
END_IF

SUPER^();

METHOD PROTECTED OnObjectStateChanged
CASE (tState) OF
	TCOM_STATE.TCOM_STATE_PREOP:
		// SyncHandler:
		RequestSyncHandlers(0, 1);
		
		// Properties:
		EnableProperty(E_BACnetPropIdentifier.PropResolution, FALSE);
		EnableProperty(E_BACnetPropIdentifier.PropScaleOffset, FALSE);

	TCOM_STATE.TCOM_STATE_SAFEOP:
		SyncProperty(E_BACnetPropIdentifier.PropPresentValue, SIZEOF(fPresentValue), ADR(fPresentValue), 0, eFullSync_InitPLC, TRUE);
		
	TCOM_STATE.TCOM_STATE_OP:
		;

END_CASE

SUPER^.OnObjectStateChanged();
END_METHOD

END_FUNCTION_BLOCK

// POUs/Local/Objects/FB_BACnet_AI_IO
// Analog Input Object
// - Terminal communication
FUNCTION_BLOCK FB_BACnet_AI_IO EXTENDS FB_BACnet_BaseAI
VAR_INPUT CONSTANT PERSISTENT	
	{region 'Variable Parameters'}
		{attribute 'parameterCategory':='Hardware'}
		fResolution : REAL := 0.1;
		{attribute 'parameterCategory':='Hardware'}
		fScaleOffset : REAL := 0;
	{endregion}
END_VAR
VAR
	{region 'Raw I/O'}
		nRawState			AT %I*	: USINT;			// Bus terminal state
		nRawValue			AT %I*	: INT;				// Bus terminal value
	{endregion}
END_VAR

SUPER^();

METHOD PROTECTED OnObjectStateChanged
CASE (tState) OF
	TCOM_STATE.TCOM_STATE_PREOP:
		// SyncHandler:
		RequestSyncHandlers(1, 4);

	TCOM_STATE.TCOM_STATE_SAFEOP:
		SyncProperty(E_BACnetPropIdentifier.PropPresentValue, SIZEOF(fPresentValue), ADR(fPresentValue), 0, eSync_FromSupplement, TRUE);
		
		SyncProperty(E_BACnetPropIdentifier.PropRawIoStateUSINT, SIZEOF(nRawState), ADR(nRawState), 0, eSync_ToSupplement, TRUE);
		SyncProperty(E_BACnetPropIdentifier.PropRawIoAnalogValueINT, SIZEOF(nRawValue), ADR(nRawValue), 0, eSync_ToSupplement, TRUE);
		
	TCOM_STATE.TCOM_STATE_OP:
		SyncProperty(E_BACnetPropIdentifier.PropResolution, SIZEOF(fResolution), ADR(fResolution), 0, eFullSync_InitPLC, FALSE);
		SyncProperty(E_BACnetPropIdentifier.PropScaleOffset, SIZEOF(fScaleOffset), ADR(fScaleOffset), 0, eFullSync_InitPLC, FALSE);

END_CASE

SUPER^.OnObjectStateChanged();
END_METHOD

END_FUNCTION_BLOCK

// POUs/Local/Objects/FB_BACnet_AI_Raw
// Analog Input Object
// - Raw communication
FUNCTION_BLOCK FB_BACnet_AI_Raw EXTENDS FB_BACnet_BaseAI
VAR_INPUT
	nRawState					: USINT;			// Raw state
													// - Underrange:	0x01
													// - Overrange:		0x02
													// - Error:			0x04
	nRawValue					: INT;				// Raw value
END_VAR
VAR_INPUT CONSTANT PERSISTENT
	{region 'Variable Parameters'}
		{attribute 'parameterCategory':='Hardware'}
		fResolution : REAL := 0.1;
		{attribute 'parameterCategory':='Hardware'}
		fScaleOffset : REAL := 0
	{endregion};
END_VAR

SUPER^();

METHOD PROTECTED OnObjectStateChanged
CASE (tState) OF
	TCOM_STATE.TCOM_STATE_PREOP:
		// SyncHandler:
		RequestSyncHandlers(1, 4);

	TCOM_STATE.TCOM_STATE_SAFEOP:
		SyncProperty(E_BACnetPropIdentifier.PropPresentValue, SIZEOF(fPresentValue), ADR(fPresentValue), 0, eSync_FromSupplement, TRUE);
		
		SyncProperty(E_BACnetPropIdentifier.PropRawIoStateUSINT, SIZEOF(nRawState), ADR(nRawState), 0, eSync_ToSupplement, TRUE);
		SyncProperty(E_BACnetPropIdentifier.PropRawIoAnalogValueINT, SIZEOF(nRawValue), ADR(nRawValue), 0, eSync_ToSupplement, TRUE);
		
	TCOM_STATE.TCOM_STATE_OP:
		SyncProperty(E_BACnetPropIdentifier.PropResolution, SIZEOF(fResolution), ADR(fResolution), 0, eFullSync_InitPLC, FALSE);
		SyncProperty(E_BACnetPropIdentifier.PropScaleOffset, SIZEOF(fScaleOffset), ADR(fScaleOffset), 0, eFullSync_InitPLC, FALSE);

END_CASE


SUPER^.OnObjectStateChanged();
END_METHOD

END_FUNCTION_BLOCK

// POUs/Local/Objects/FB_BACnet_AV_Disp
// Analog Setpoint Object for Operation
// - Used to display a value
FUNCTION_BLOCK FB_BACnet_AV_Disp EXTENDS FB_BACnet_Object
VAR_INPUT
	fVal			: REAL;
END_VAR
VAR_INPUT CONSTANT PERSISTENT
	{region 'Variable Parameters'}
		{attribute 'parameterCategory':='Value'}
		fCOVIncrement : REAL := 0.1;
		{attribute 'parameterCategory':='Value'}
		eUnit : E_BA_Unit := E_BA_Unit.eOther_NoUnits;
	{endregion}
END_VAR
VAR_OUTPUT
	fPresentValue	: REAL;
END_VAR

IF bReady THEN
	fPresentValue := fVal;
ELSE
	fPresentValue := 0;
END_IF

SUPER^();

METHOD PROTECTED OnObjectStateChanged
SUPER^.OnObjectStateChanged();

CASE (tState) OF
	TCOM_STATE.TCOM_STATE_PREOP:
		// SyncHandler:
		RequestSyncHandlers(0, 3);
		
		// Properties:
		// EnableProperty(E_BACnetPropIdentifier.PropDeviceType, FALSE);
		EnableProperty(E_BACnetPropIdentifier.PropNotificationClass, FALSE);
		EnableProperty(E_BACnetPropIdentifier.PropNotifyType, FALSE);
		EnableProperty(E_BACnetPropIdentifier.PropEventEnable, FALSE);
		EnableProperty(E_BACnetPropIdentifier.PropEventTimeStamps, FALSE);
		EnableProperty(E_BACnetPropIdentifier.PropEventMessageTexts, FALSE);
		EnableProperty(E_BACnetPropIdentifier.PropEventMessageTextsConfig, FALSE);
		EnableProperty(E_BACnetPropIdentifier.PropTimeDelay, FALSE);
		EnableProperty(E_BACnetPropIdentifier.PropStatusFlags, FALSE);
		EnableProperty(E_BACnetPropIdentifier.PropAckedTransitions, FALSE);
		EnableProperty(E_BACnetPropIdentifier.PropReliability, FALSE);
		EnableProperty(E_BACnetPropIdentifier.PropEventState, FALSE);
		EnableProperty(E_BACnetPropIdentifier.PropEventDetectionEnable, FALSE);
		EnableProperty(E_BACnetPropIdentifier.PropEventAlgorithmInhibit, FALSE);
		EnableProperty(E_BACnetPropIdentifier.PropTimeDelayNormal, FALSE);
		EnableProperty(E_BACnetPropIdentifier.PropReliabilityEvaluationInhibit, FALSE);
		EnableProperty(E_BACnetPropIdentifier.PropLimitEnable, FALSE);
		EnableProperty(E_BACnetPropIdentifier.PropHighLimit, FALSE);
		EnableProperty(E_BACnetPropIdentifier.PropLowLimit, FALSE);
		EnableProperty(E_BACnetPropIdentifier.PropDeadband, FALSE);
		EnableProperty(E_BACnetPropIdentifier.PropRelinquishDefault, FALSE);
		EnableProperty(E_BACnetPropIdentifier.PropPriorityArray, FALSE);
		EnableProperty(E_BACnetPropIdentifier.PropOutOfService, FALSE);
		EnableProperty(E_BACnetPropIdentifier.PropCurrentlyActivePriority, FALSE);
		
		WriteProtectProperty(E_BACnetPropIdentifier.PropPresentValue, TRUE);
		
	TCOM_STATE.TCOM_STATE_SAFEOP:
		SyncProperty(E_BACnetPropIdentifier.PropPresentValue, SIZEOF(fVal), ADR(fVal), 0, eSync_ToSupplement, TRUE);
		
	TCOM_STATE.TCOM_STATE_OP:
		SyncProperty(E_BACnetPropIdentifier.PropUnits, SIZEOF(eUnit), ADR(eUnit), 0, eFullSync_InitPLC, FALSE);
		SyncProperty(E_BACnetPropIdentifier.PropCovIncrement, SIZEOF(fCOVIncrement), ADR(fCOVIncrement), 0, eFullSync_InitPLC, FALSE);
END_CASE
END_METHOD

METHOD FB_init : BOOL
VAR_INPUT
	bInitRetains : BOOL; // if TRUE, the retain variables are initialized (warm start / cold start)
	bInCopyCode : BOOL;  // if TRUE, the instance afterwards gets moved into the copy code (online change)
END_VAR
eObjectType := E_BACnetObjType.ObjAnalogValue;
END_METHOD

END_FUNCTION_BLOCK

// POUs/Local/Objects/FB_BACnet_AV_Setp
// Analog Setpoint Object for Operation
// - Used to define a setpoint by user
FUNCTION_BLOCK FB_BACnet_AV_Setp EXTENDS FB_BACnet_Object
VAR_INPUT CONSTANT PERSISTENT
	{region 'Variable Parameters'}
		{attribute 'parameterCategory':='Value'}
		fCOVIncrement : REAL := 0.1;
		{attribute 'parameterCategory':='Value'}
		eUnit : E_BA_Unit := E_BA_Unit.eOther_NoUnits;
	{endregion}
	{region 'Operational Parameters'}
		{attribute 'parameterCategory':='Value'}
		fValue : REAL;
	{endregion}
END_VAR
VAR_OUTPUT
	fPresentValue	: REAL;
END_VAR

IF bReady THEN
	fPresentValue := fValue;
ELSE
	fPresentValue := 0;
END_IF

SUPER^();

METHOD PROTECTED OnObjectStateChanged
SUPER^.OnObjectStateChanged();

CASE (tState) OF
	TCOM_STATE.TCOM_STATE_PREOP:
		// SyncHandler:
		RequestSyncHandlers(0, 3);
		
		// Properties:
		// DisableProperty(E_BACnetPropIdentifier.PropDeviceType, FALSE);
		EnableProperty(E_BACnetPropIdentifier.PropNotificationClass, FALSE);
		EnableProperty(E_BACnetPropIdentifier.PropNotifyType, FALSE);
		EnableProperty(E_BACnetPropIdentifier.PropEventEnable, FALSE);
		EnableProperty(E_BACnetPropIdentifier.PropEventTimeStamps, FALSE);
		EnableProperty(E_BACnetPropIdentifier.PropEventMessageTexts, FALSE);
		EnableProperty(E_BACnetPropIdentifier.PropEventMessageTextsConfig, FALSE);
		EnableProperty(E_BACnetPropIdentifier.PropTimeDelay, FALSE);
		EnableProperty(E_BACnetPropIdentifier.PropStatusFlags, FALSE);
		EnableProperty(E_BACnetPropIdentifier.PropAckedTransitions, FALSE);
		EnableProperty(E_BACnetPropIdentifier.PropReliability, FALSE);
		EnableProperty(E_BACnetPropIdentifier.PropEventState, FALSE);
		EnableProperty(E_BACnetPropIdentifier.PropEventDetectionEnable, FALSE);
		EnableProperty(E_BACnetPropIdentifier.PropEventAlgorithmInhibit, FALSE);
		EnableProperty(E_BACnetPropIdentifier.PropTimeDelayNormal, FALSE);
		EnableProperty(E_BACnetPropIdentifier.PropReliabilityEvaluationInhibit, FALSE);
		EnableProperty(E_BACnetPropIdentifier.PropLimitEnable, FALSE);
		EnableProperty(E_BACnetPropIdentifier.PropHighLimit, FALSE);
		EnableProperty(E_BACnetPropIdentifier.PropLowLimit, FALSE);
		EnableProperty(E_BACnetPropIdentifier.PropDeadband, FALSE);
		EnableProperty(E_BACnetPropIdentifier.PropRelinquishDefault, FALSE);
		EnableProperty(E_BACnetPropIdentifier.PropPriorityArray, FALSE);
		EnableProperty(E_BACnetPropIdentifier.PropOutOfService, FALSE);
		EnableProperty(E_BACnetPropIdentifier.PropCurrentlyActivePriority, FALSE);
		
	TCOM_STATE.TCOM_STATE_SAFEOP:
		;
		
	TCOM_STATE.TCOM_STATE_OP:
		SyncProperty(E_BACnetPropIdentifier.PropPresentValue, SIZEOF(fValue), ADR(fValue), 0, eFullSync_InitPLC, FALSE);
		
		SyncProperty(E_BACnetPropIdentifier.PropUnits, SIZEOF(eUnit), ADR(eUnit), 0, eFullSync_InitPLC, FALSE);
		SyncProperty(E_BACnetPropIdentifier.PropCovIncrement, SIZEOF(fCOVIncrement), ADR(fCOVIncrement), 0, eFullSync_InitPLC, FALSE);
END_CASE
END_METHOD

METHOD FB_init : BOOL
VAR_INPUT
	bInitRetains : BOOL; // if TRUE, the retain variables are initialized (warm start / cold start)
	bInCopyCode : BOOL;  // if TRUE, the instance afterwards gets moved into the copy code (online change)
END_VAR
eObjectType := E_BACnetObjType.ObjAnalogValue;
END_METHOD

END_FUNCTION_BLOCK

// POUs/Local/Objects/FB_BACnet_BI_IO
// Binary Input Object
// - Terminal communication
FUNCTION_BLOCK FB_BACnet_BI_IO EXTENDS FB_BACnet_BaseBI
VAR
	{region 'Raw I/O'}
		bRawValue			AT %I*	: BOOL;				// Bus terminal value
	{endregion}
END_VAR

SUPER^();

METHOD PROTECTED OnObjectStateChanged
SUPER^.OnObjectStateChanged();

CASE (tState) OF
	TCOM_STATE.TCOM_STATE_PREOP:
		// SyncHandler:
		RequestSyncHandlers(0, 1);

	TCOM_STATE.TCOM_STATE_SAFEOP:
		SyncProperty(E_BACnetPropIdentifier.PropRawIoBinaryValueBOOL, SIZEOF(bRawValue), ADR(bRawValue), 0, eSync_ToSupplement, TRUE);
		
	TCOM_STATE.TCOM_STATE_OP:
		;

END_CASE
END_METHOD

END_FUNCTION_BLOCK

// POUs/Local/Objects/FB_BACnet_BI_Raw
// Binary Input Object
// - Raw communication
FUNCTION_BLOCK FB_BACnet_BI_Raw EXTENDS FB_BACnet_BaseBI
VAR_INPUT
	bRawValue					: BOOL;				// Raw value
END_VAR

SUPER^();

METHOD PROTECTED OnObjectStateChanged
SUPER^.OnObjectStateChanged();

CASE (tState) OF
	TCOM_STATE.TCOM_STATE_PREOP:
		// SyncHandler:
		RequestSyncHandlers(0, 1);

	TCOM_STATE.TCOM_STATE_SAFEOP:
		SyncProperty(E_BACnetPropIdentifier.PropRawIoBinaryValueBOOL, SIZEOF(bRawValue), ADR(bRawValue), 0, eSync_ToSupplement, TRUE);
		
	TCOM_STATE.TCOM_STATE_OP:
		;

END_CASE
END_METHOD

END_FUNCTION_BLOCK

// POUs/Local/Objects/FB_BACnet_BV_Disp
// Binary Setpoint Object for Operation
// - Used to display a value
FUNCTION_BLOCK FB_BACnet_BV_Disp EXTENDS FB_BACnet_Object
VAR_INPUT
	bVal			: BOOL;
END_VAR
VAR_INPUT CONSTANT PERSISTENT
	{region 'Variable Parameters'}
		{attribute 'parameterCategory':='Value'}
		{attribute 'TcEncoding':='UTF-8'}
		sInactiveText : T_BACnet_StateText;
		{attribute 'parameterCategory':='Value'}
		{attribute 'TcEncoding':='UTF-8'}
		sActiveText : T_BACnet_StateText;
	{endregion}
END_VAR
VAR_OUTPUT
	bPresentValue	: BOOL;
END_VAR

IF bReady THEN
	bPresentValue := bVal;
ELSE
	bPresentValue := FALSE;
END_IF

SUPER^();

METHOD PROTECTED OnObjectStateChanged
SUPER^.OnObjectStateChanged();

CASE (tState) OF
	TCOM_STATE.TCOM_STATE_PREOP:
		// SyncHandler:
		RequestSyncHandlers(0, 3);
		
		// Properties:
		EnableProperty(E_BACnetPropIdentifier.PropDeviceType, FALSE);
		EnableProperty(E_BACnetPropIdentifier.PropMinimumOnTime, FALSE);
		EnableProperty(E_BACnetPropIdentifier.PropMinimumOffTime, FALSE);
		EnableProperty(E_BACnetPropIdentifier.PropNotificationClass, FALSE);
		EnableProperty(E_BACnetPropIdentifier.PropNotifyType, FALSE);
		EnableProperty(E_BACnetPropIdentifier.PropEventEnable, FALSE);
		EnableProperty(E_BACnetPropIdentifier.PropEventTimeStamps, FALSE);
		EnableProperty(E_BACnetPropIdentifier.PropEventMessageTexts, FALSE);
		EnableProperty(E_BACnetPropIdentifier.PropEventMessageTextsConfig, FALSE);
		EnableProperty(E_BACnetPropIdentifier.PropTimeDelay, FALSE);
		EnableProperty(E_BACnetPropIdentifier.PropStatusFlags, FALSE);
		EnableProperty(E_BACnetPropIdentifier.PropAckedTransitions, FALSE);
		EnableProperty(E_BACnetPropIdentifier.PropReliability, FALSE);
		EnableProperty(E_BACnetPropIdentifier.PropEventState, FALSE);
		EnableProperty(E_BACnetPropIdentifier.PropEventDetectionEnable, FALSE);
		EnableProperty(E_BACnetPropIdentifier.PropEventAlgorithmInhibit, FALSE);
		EnableProperty(E_BACnetPropIdentifier.PropTimeDelayNormal, FALSE);
		EnableProperty(E_BACnetPropIdentifier.PropReliabilityEvaluationInhibit, FALSE);
		EnableProperty(E_BACnetPropIdentifier.PropChangeOfStateCount, FALSE);
		EnableProperty(E_BACnetPropIdentifier.PropChangeOfStateTime, FALSE);
		EnableProperty(E_BACnetPropIdentifier.PropTimeOfStateCountReset, FALSE);
		EnableProperty(E_BACnetPropIdentifier.PropElapsedActiveTime, FALSE);
		EnableProperty(E_BACnetPropIdentifier.PropTimeOfActiveTimeReset, FALSE);
		EnableProperty(E_BACnetPropIdentifier.PropRelinquishDefault, FALSE);
		EnableProperty(E_BACnetPropIdentifier.PropPriorityArray, FALSE);
		EnableProperty(E_BACnetPropIdentifier.PropOutOfService, FALSE);
		EnableProperty(E_BACnetPropIdentifier.PropCurrentlyActivePriority, FALSE);
		
		WriteProtectProperty(E_BACnetPropIdentifier.PropPresentValue, TRUE);
		
		IF (BACnet_Param.bStateText_WriteProtect) THEN
			WriteProtectProperty(E_BACnetPropIdentifier.PropActiveText, TRUE);
			WriteProtectProperty(E_BACnetPropIdentifier.PropInactiveText, TRUE);
		END_IF
		
		// Ensure UTF-8 Encoding:
		F_BA_EnsureUTF8(ADR(sInactiveText), SIZEOF(sInactiveText));
		F_BA_EnsureUTF8(ADR(sActiveText), SIZEOF(sActiveText));
		
	TCOM_STATE.TCOM_STATE_SAFEOP:
		SyncProperty(E_BACnetPropIdentifier.PropPresentValue, SIZEOF(bVal), ADR(bVal), 0, eSync_ToSupplement, TRUE);
		
	TCOM_STATE.TCOM_STATE_OP:
		SyncProperty(E_BACnetPropIdentifier.PropActiveText, SIZEOF(sActiveText), ADR(sActiveText), 0, eFullSync_InitPLC, FALSE);	
		SyncProperty(E_BACnetPropIdentifier.PropInactiveText, SIZEOF(sInactiveText), ADR(sInactiveText), 0, eFullSync_InitPLC, FALSE);
END_CASE
END_METHOD

METHOD FB_init : BOOL
VAR_INPUT
	bInitRetains : BOOL; // if TRUE, the retain variables are initialized (warm start / cold start)
	bInCopyCode : BOOL;  // if TRUE, the instance afterwards gets moved into the copy code (online change)
END_VAR
eObjectType := E_BACnetObjType.ObjBinaryValue;
END_METHOD

END_FUNCTION_BLOCK

// POUs/Local/Objects/FB_BACnet_BV_Setp
// Binary Setpoint Object for Operation
// - Used to define a setpoint by user
FUNCTION_BLOCK FB_BACnet_BV_Setp EXTENDS FB_BACnet_Object
VAR_INPUT CONSTANT PERSISTENT
	{region 'Variable Parameters'}
		{attribute 'parameterCategory':='Value'}
		{attribute 'TcEncoding':='UTF-8'}
		sInactiveText : T_BACnet_StateText;
		{attribute 'parameterCategory':='Value'}
		{attribute 'TcEncoding':='UTF-8'}
		sActiveText : T_BACnet_StateText;
	{endregion}
	{region 'Operational Parameters'}
		{attribute 'parameterCategory':='Value'}
		bValue : BOOL;
	{endregion}
END_VAR
VAR_OUTPUT
	bPresentValue	: BOOL;
END_VAR

IF bReady THEN
	bPresentValue := bValue;
ELSE
	bPresentValue := FALSE;
END_IF

SUPER^();

METHOD PROTECTED OnObjectStateChanged
SUPER^.OnObjectStateChanged();

CASE (tState) OF
	TCOM_STATE.TCOM_STATE_PREOP:
		// SyncHandler:
		RequestSyncHandlers(0, 3);
		
		// Properties:
		EnableProperty(E_BACnetPropIdentifier.PropDeviceType, FALSE);
		EnableProperty(E_BACnetPropIdentifier.PropMinimumOnTime, FALSE);
		EnableProperty(E_BACnetPropIdentifier.PropMinimumOffTime, FALSE);
		EnableProperty(E_BACnetPropIdentifier.PropNotificationClass, FALSE);
		EnableProperty(E_BACnetPropIdentifier.PropNotifyType, FALSE);
		EnableProperty(E_BACnetPropIdentifier.PropEventEnable, FALSE);
		EnableProperty(E_BACnetPropIdentifier.PropEventTimeStamps, FALSE);
		EnableProperty(E_BACnetPropIdentifier.PropEventMessageTexts, FALSE);
		EnableProperty(E_BACnetPropIdentifier.PropEventMessageTextsConfig, FALSE);
		EnableProperty(E_BACnetPropIdentifier.PropTimeDelay, FALSE);
		EnableProperty(E_BACnetPropIdentifier.PropStatusFlags, FALSE);
		EnableProperty(E_BACnetPropIdentifier.PropAckedTransitions, FALSE);
		EnableProperty(E_BACnetPropIdentifier.PropReliability, FALSE);
		EnableProperty(E_BACnetPropIdentifier.PropEventState, FALSE);
		EnableProperty(E_BACnetPropIdentifier.PropEventDetectionEnable, FALSE);
		EnableProperty(E_BACnetPropIdentifier.PropEventAlgorithmInhibit, FALSE);
		EnableProperty(E_BACnetPropIdentifier.PropTimeDelayNormal, FALSE);
		EnableProperty(E_BACnetPropIdentifier.PropReliabilityEvaluationInhibit, FALSE);
		EnableProperty(E_BACnetPropIdentifier.PropChangeOfStateCount, FALSE);
		EnableProperty(E_BACnetPropIdentifier.PropChangeOfStateTime, FALSE);
		EnableProperty(E_BACnetPropIdentifier.PropTimeOfStateCountReset, FALSE);
		EnableProperty(E_BACnetPropIdentifier.PropElapsedActiveTime, FALSE);
		EnableProperty(E_BACnetPropIdentifier.PropTimeOfActiveTimeReset, FALSE);
		EnableProperty(E_BACnetPropIdentifier.PropRelinquishDefault, FALSE);
		EnableProperty(E_BACnetPropIdentifier.PropPriorityArray, FALSE);
		EnableProperty(E_BACnetPropIdentifier.PropOutOfService, FALSE);
		EnableProperty(E_BACnetPropIdentifier.PropCurrentlyActivePriority, FALSE);
		
		IF (BACnet_Param.bStateText_WriteProtect) THEN
			WriteProtectProperty(E_BACnetPropIdentifier.PropActiveText, TRUE);
			WriteProtectProperty(E_BACnetPropIdentifier.PropInactiveText, TRUE);
		END_IF
		
		// Ensure UTF-8 Encoding:
		F_BA_EnsureUTF8(ADR(sInactiveText), SIZEOF(sInactiveText));
		F_BA_EnsureUTF8(ADR(sActiveText), SIZEOF(sActiveText));
		
	TCOM_STATE.TCOM_STATE_SAFEOP:
		;
		
	TCOM_STATE.TCOM_STATE_OP:
		SyncProperty(E_BACnetPropIdentifier.PropPresentValue, SIZEOF(bValue), ADR(bValue), 0, eFullSync_InitPLC, FALSE);
		
		SyncProperty(E_BACnetPropIdentifier.PropActiveText, SIZEOF(sActiveText), ADR(sActiveText), 0, eFullSync_InitPLC, FALSE);	
		SyncProperty(E_BACnetPropIdentifier.PropInactiveText, SIZEOF(sInactiveText), ADR(sInactiveText), 0, eFullSync_InitPLC, FALSE);
END_CASE
END_METHOD

METHOD FB_init : BOOL
VAR_INPUT
	bInitRetains : BOOL; // if TRUE, the retain variables are initialized (warm start / cold start)
	bInCopyCode : BOOL;  // if TRUE, the instance afterwards gets moved into the copy code (online change)
END_VAR
eObjectType := E_BACnetObjType.ObjBinaryValue;
END_METHOD

END_FUNCTION_BLOCK

// POUs/Local/Objects/FB_BACnet_Cal
// Calendar Object
FUNCTION_BLOCK FB_BACnet_Cal EXTENDS FB_BACnet_Object IMPLEMENTS I_BACnet_Cal
VAR_INPUT CONSTANT PERSISTENT
	{region 'Variable Parameters'}
		{attribute 'parameterCategory':='Value'}
		tDateList : T_BACnet_CalendarDateList;
	{endregion}
END_VAR
VAR_INPUT CONSTANT
	{region 'Variable Parameters'}
		{attribute 'parameterCategory':='Value'}
		bWriteDateList : BOOL;
	{endregion}
END_VAR
VAR_OUTPUT
	bPresentValue			: BOOL;
END_VAR
VAR	
	{region 'COV'}
		bDateListChanged	: BOOL;
	{endregion}
END_VAR

IF (bWriteDateList) THEN
	WriteContent();
	bWriteDateList := FALSE;
END_IF
IF (bDateListChanged) THEN
	ReadContent();
	bDateListChanged := FALSE;
END_IF

SUPER^();

METHOD PROTECTED OnObjectStateChanged
SUPER^.OnObjectStateChanged();

CASE (tState) OF
	TCOM_STATE.TCOM_STATE_PREOP:
		// SyncHandler:
		RequestSyncHandlers(2, 0);

	TCOM_STATE.TCOM_STATE_SAFEOP:
		;
		
	TCOM_STATE.TCOM_STATE_OP:
		SyncProperty(E_BACnetPropIdentifier.PropPresentValue, SIZEOF(bPresentValue), ADR(bPresentValue), 0, eSync_FromSupplement, FALSE);
		
		SyncPropertyCOV(bDateListChanged, E_BACnetPropIdentifier.PropDateList);
	
		WriteContent();
		
END_CASE
END_METHOD

METHOD FB_init : BOOL
VAR_INPUT
	bInitRetains : BOOL; // if TRUE, the retain variables are initialized (warm start / cold start)
	bInCopyCode : BOOL;  // if TRUE, the instance afterwards gets moved into the copy code (online change)
END_VAR
eObjectType := E_BACnetObjType.ObjCalendar;
END_METHOD

METHOD ReadContent : BOOL
ReadContent := (ReadPropertyDateList(tDateList) = S_OK);
END_METHOD

METHOD WriteContent : BOOL
WriteContent := (WritePropertyDateList(tDateList) = S_OK);
END_METHOD

END_FUNCTION_BLOCK

// POUs/Local/Objects/FB_BACnet_Device
// Device Object
FUNCTION_BLOCK FB_BACnet_Device EXTENDS FB_BACnet_Object
VAR_INPUT CONSTANT PERSISTENT
	{region 'Variable Parameters'}
		{attribute 'parameterCategory':='Communication'}
		{attribute 'parameterUnit':= 'ms'}
		nAPDUSegmentTimeout : UDINT := 2000;						// (in [ms])
		{attribute 'parameterCategory':='Communication'}
		{attribute 'parameterUnit':= 'ms'}
		nAPDUTimeout : UDINT := 3000;								// (in [ms])
		{attribute 'parameterCategory':='Communication'}
		nNumberOfAPDURetries : UDINT := 3;
			 
		{attribute 'parameterCategory':='General'}
		{attribute 'TcEncoding':='UTF-8'}
		sLocation : T_MaxString;
	{endregion}
END_VAR
VAR_OUTPUT
	dtLocalTime			: ST_BA_DateTime;
END_VAR

SUPER^();

METHOD PROTECTED OnObjectStateChanged
SUPER^.OnObjectStateChanged();

CASE (tState) OF
	TCOM_STATE.TCOM_STATE_PREOP:
		// SyncHandler:
		RequestSyncHandlers(2, 4);
		
		// Ensure UTF-8 Encoding:
		F_BA_EnsureUTF8(ADR(sLocation), SIZEOF(sLocation));
		
	TCOM_STATE.TCOM_STATE_SAFEOP:
		;
	
	TCOM_STATE.TCOM_STATE_OP:
		SyncProperty(E_BACnetPropIdentifier.PropLocalTime, SIZEOF(dtLocalTime.stTime), ADR(dtLocalTime.stTime), 0, eSync_FromSupplement, FALSE);
		SyncProperty(E_BACnetPropIdentifier.PropLocalDate, SIZEOF(dtLocalTime.stDate), ADR(dtLocalTime.stDate), 0, eSync_FromSupplement, FALSE);
		
		SyncProperty(E_BACnetPropIdentifier.PropApduSegmentTimeout, SIZEOF(nAPDUSegmentTimeout), ADR(nAPDUSegmentTimeout), 0, eFullSync_InitPLC, FALSE);
		SyncProperty(E_BACnetPropIdentifier.PropApduTimeout, SIZEOF(nAPDUTimeout), ADR(nAPDUTimeout), 0, eFullSync_InitPLC, FALSE);
		SyncProperty(E_BACnetPropIdentifier.PropNumberOfAPDURetries, SIZEOF(nNumberOfAPDURetries), ADR(nNumberOfAPDURetries), 0, eFullSync_InitPLC, FALSE);
		SyncProperty(E_BACnetPropIdentifier.PropLocation, SIZEOF(sLocation), ADR(sLocation), 0, eFullSync_InitPLC, FALSE);
		
END_CASE
END_METHOD

METHOD FB_init : BOOL
VAR_INPUT
	bInitRetains : BOOL; // if TRUE, the retain variables are initialized (warm start / cold start)
	bInCopyCode : BOOL;  // if TRUE, the instance afterwards gets moved into the copy code (online change)
END_VAR
eObjectType := E_BACnetObjType.ObjDevice;
END_METHOD

PROPERTY Location : T_MaxString
GET
Location:=sLocation;
END_GET
SET
sLocation:=Location;
END_SET
END_PROPERTY

END_FUNCTION_BLOCK

// POUs/Local/Objects/FB_BACnet_EventLog
// Event Log Object
FUNCTION_BLOCK FB_BACnet_EventLog EXTENDS FB_BACnet_Object
VAR_INPUT CONSTANT PERSISTENT
	{region 'Fixed Parameters'}
		{attribute 'parameterCategory':='Value'}
		nBufferSize : UDINT := BACnet_Param.nEventLog_ArraySize;
		// (BETA) ... Implement "EventLogBuffer"-Property
		//{attribute 'hide'}
		//{attribute 'parameterCategory':='Value'}
		//tLogBuffer : ARRAY [1 .. BACnet_Param.nEventLog_ArraySize] OF ST_BACnet_EventLogEntry;
			 
		{attribute 'parameterCategory':='Config'}
		nProcessId : UDINT;
	{endregion}
	{region 'Variable Parameters'}
		{attribute 'parameterCategory':='State'}
		bLogEnable : BOOL;
			 
		{attribute 'parameterCategory':='EventConfig'}
		nNotificationClass : UDINT;
		{attribute 'parameterCategory':='EventConfig'}
		eNotifyType : E_BACnet_NotifyType := E_BACnet_NotifyType.eAlarm;
		{attribute 'parameterCategory':='EventConfig'}
		bEventEnable : ARRAY[E_BA_EventTransition.First .. E_BA_EventTransition.Last] OF BOOL;
		{attribute 'parameterCategory':='EventConfig'}
		sEventMessageTextsConfig : ARRAY[E_BA_EventTransition.First .. E_BA_EventTransition.Last] OF T_MaxString;
		
		{attribute 'parameterCategory':='Config'}
		stStartTime : ST_BA_DateTime;
		{attribute 'parameterCategory':='Config'}
		stStopTime : ST_BA_DateTime;
		{attribute 'parameterCategory':='Config'}
		bStopWhenFull : BOOL;
		{attribute 'parameterCategory':='Config'}
		nNotificationThreshold : UDINT := 50;
	{endregion}
END_VAR
VAR_OUTPUT
	nRecordCount				: UDINT;
	nTotalRecordCount			: UDINT;
END_VAR
VAR
	{region 'Buffers'}
		{attribute 'hide'}
		fbLogBuffer				: FB_BACnet_EventLogBuffer	:= (iRefObject := THIS^);
	{endregion}
END_VAR

// Synchronize Buffers:
fbLogBuffer();

SUPER^();

METHOD PROTECTED OnObjectStateChanged
SUPER^.OnObjectStateChanged();

// Synchronize:
fbLogBuffer.OnObjectStateChanged(tState);

CASE (tState) OF
	TCOM_STATE.TCOM_STATE_PREOP:
		// SyncHandler:
		RequestSyncHandlers(2, 14);
		
		// Properties:
		// May limit buffer size to respect array size:
		nBufferSize := MIN(BACnet_Param.nEventLog_ArraySize, nBufferSize);
		
		WritePropertyUDInt(E_BACnetPropIdentifier.PropBufferSize, nBufferSize);
		
		// Ensure UTF-8 Encoding:
		F_BA_EnsureUTF8Array(ADR(sEventMessageTextsConfig), SIZEOF(sEventMessageTextsConfig[1]), TO_DINT(E_BA_EventTransition.Count));
		
	TCOM_STATE.TCOM_STATE_SAFEOP:
		;

	TCOM_STATE.TCOM_STATE_OP:
		ConcatTitle(sEventMessageTextsConfig[E_BA_EventTransition.eToOffnormal], sDescription, BACnet_Param.sSeparator_EventMessageText);
		ConcatTitle(sEventMessageTextsConfig[E_BA_EventTransition.eToFault], sDescription, BACnet_Param.sSeparator_EventMessageText);
		ConcatTitle(sEventMessageTextsConfig[E_BA_EventTransition.eToNormal], sDescription, BACnet_Param.sSeparator_EventMessageText);
		
		// Synchronize:
		SyncProperty(E_BACnetPropIdentifier.PropRecordCount, SIZEOF(nRecordCount), ADR(nRecordCount), 0, eSync_FromSupplement, FALSE);
		SyncProperty(E_BACnetPropIdentifier.PropTotalRecordCount, SIZEOF(nTotalRecordCount), ADR(nTotalRecordCount), 0, eSync_FromSupplement, FALSE);
		
		SyncProperty(E_BACnetPropIdentifier.PropNotificationClass, SIZEOF(nNotificationClass), ADR(nNotificationClass), 0, eFullSync_InitPLC, FALSE);
		SyncProperty(E_BACnetPropIdentifier.PropNotifyType, SIZEOF(eNotifyType), ADR(eNotifyType), 0, eFullSync_InitPLC, FALSE);
		SyncPropertyIdx(E_BACnetPropIdentifier.PropEventEnable, SIZEOF(BOOL), ADR(bEventEnable[E_BA_EventTransition.eToOffnormal]), E_BACnet_EventTransitionBits.eToOffnormal, 0, eFullSync_InitPLC, FALSE);	
		SyncPropertyIdx(E_BACnetPropIdentifier.PropEventEnable, SIZEOF(BOOL), ADR(bEventEnable[E_BA_EventTransition.eToFault]), E_BACnet_EventTransitionBits.eToFault, 0, eFullSync_InitPLC, FALSE);	
		SyncPropertyIdx(E_BACnetPropIdentifier.PropEventEnable, SIZEOF(BOOL), ADR(bEventEnable[E_BA_EventTransition.eToNormal]), E_BACnet_EventTransitionBits.eToNormal, 0, eFullSync_InitPLC, FALSE);
		SyncPropertyIdx(E_BACnetPropIdentifier.PropEventMessageTextsConfig, SIZEOF(T_MaxString), ADR(sEventMessageTextsConfig[E_BA_EventTransition.eToOffnormal]), (E_BACnet_EventTransitionBits.eToOffnormal+1), 0, eFullSync_InitPLC, FALSE);
		SyncPropertyIdx(E_BACnetPropIdentifier.PropEventMessageTextsConfig, SIZEOF(T_MaxString), ADR(sEventMessageTextsConfig[E_BA_EventTransition.eToFault]), (E_BACnet_EventTransitionBits.eToFault+1), 0, eFullSync_InitPLC, FALSE);
		SyncPropertyIdx(E_BACnetPropIdentifier.PropEventMessageTextsConfig, SIZEOF(T_MaxString), ADR(sEventMessageTextsConfig[E_BA_EventTransition.eToNormal]), (E_BACnet_EventTransitionBits.eToNormal+1), 0, eFullSync_InitPLC, FALSE);
		
		SyncProperty(E_BACnetPropIdentifier.PropEnable, SIZEOF(bLogEnable), ADR(bLogEnable), 0, eFullSync_InitPLC, FALSE);
		SyncProperty(E_BACnetPropIdentifier.PropStartTime, SIZEOF(stStartTime), ADR(stStartTime), 0, eFullSync_InitPLC, FALSE);
		SyncProperty(E_BACnetPropIdentifier.PropStopTime, SIZEOF(stStopTime), ADR(stStopTime), 0, eFullSync_InitPLC, FALSE);
		SyncProperty(E_BACnetPropIdentifier.PropStopWhenFull, SIZEOF(bStopWhenFull), ADR(bStopWhenFull), 0, eFullSync_InitPLC, FALSE);
		SyncProperty(E_BACnetPropIdentifier.PropNotificationThreshold, SIZEOF(nNotificationThreshold), ADR(nNotificationThreshold), 0, eFullSync_InitPLC, FALSE);
		SyncProperty(E_BACnetPropIdentifier.PropProcessId, SIZEOF(nProcessId), ADR(nProcessId), 0, eFullSync_InitPLC, FALSE);
		
END_CASE
END_METHOD

METHOD FB_init : BOOL
VAR_INPUT
	bInitRetains : BOOL; // if TRUE, the retain variables are initialized (warm start / cold start)
	bInCopyCode : BOOL;  // if TRUE, the instance afterwards gets moved into the copy code (online change)
END_VAR
eObjectType := E_BACnetObjType.ObjEventLog;
END_METHOD

END_FUNCTION_BLOCK

// POUs/Local/Objects/FB_BACnet_Loop
// Loop Object
FUNCTION_BLOCK FB_BACnet_Loop EXTENDS FB_BACnet_EventObject
VAR_INPUT
	bEn						: BOOL;
	fSetpoint				: REAL;
	fCtrlVar				: REAL;

	bEnSync					: BOOL;
	fValSync				: REAL;
END_VAR
VAR_INPUT CONSTANT PERSISTENT
	{region 'Variable Parameters'}
		{attribute 'parameterCategory':='Value'}
		bEnOutOfService : BOOL;
		{attribute 'parameterCategory':='Value'}
		fCOVIncrement : REAL := 0.1;
		{attribute 'parameterCategory':='Value'}
		eOutputUnit : E_BA_Unit := E_BA_Unit.eOther_Percent;
		
		{attribute 'parameterCategory':='Config'}
		eAction : E_BA_Action := E_BA_Action.eDirect;
		{attribute 'parameterCategory':='Config'}
		fBias : REAL := 0;
		{attribute 'parameterCategory':='Config'}
		fMinOutput : REAL := 0;
		{attribute 'parameterCategory':='Config'}
		fMaxOutput : REAL := 100;
		{attribute 'parameterCategory':='Config'}
		fAccLimit : REAL := 0.0;							// Setpoint acceleration limit positive and negative [1/s]
		{attribute 'parameterCategory':='Config'}
		fPropertionalConstant : REAL := 1;
		{attribute 'parameterCategory':='Config'}
		ePropertionalConstantUnit : E_BA_Unit := E_BA_Unit.eOther_NoUnits;
		{attribute 'parameterCategory':='Config'}
		fIntegralConstant : REAL := 60;
		{attribute 'parameterCategory':='Config'}
		eIntegralConstantUnit : E_BA_Unit := E_BA_Unit.eTime_Seconds;
		{attribute 'parameterCategory':='Config'}
		fDerivativeConstant : REAL := 0;
		{attribute 'parameterCategory':='Config'}
		eDerivativeConstantUnit : E_BA_Unit := E_BA_Unit.eTime_Seconds;
		
		{attribute 'parameterCategory':='EventConfig'}
		fDeadband : REAL := 0.1;
		{attribute 'parameterCategory':='EventConfig'}
		fErrorLimit : REAL := 0;
	{endregion}
END_VAR
VAR_OUTPUT
	fPresentValue			: REAL;
END_VAR
VAR
	{region 'Output-Properties'}
		eMode				: E_BACnet_LoopMode;
		fPropBand			: REAL; 						// Controller output in range of -100...100% in relation to Min.-/Max.-output
	{endregion}
END_VAR
VAR
	{region 'Internal'}
		{attribute 'hide'}
		fbIntCtrl			: FB_BACnet_PidControl;
		{attribute 'hide'}
		fbAccLimit			: FB_BACnet_AccLimit;
	{endregion}
	{region 'Temporary'}
		{attribute 'hide'}
		_sysTime			: GETCPUCOUNTER;
		{attribute 'hide'}
		_Time				: T_LARGE_INTEGER;
		{attribute 'hide'}
		_TimeOld			: T_LARGE_INTEGER;
		{attribute 'hide'}
		_tCycleTime			: REAL;
	{endregion}
END_VAR

IF (bReady) THEN
	// Determine cycle time:
	_TimeOld := _Time;
	_sysTime(cpuCntLoDW=>_Time.dwLowPart, cpuCntHiDW=>_Time.dwHighPart);
	_tCycleTime := F_BACnet_SysTimeDiff(In1:=_Time, In2:=_TimeOld);

	// Check PID mode:
	IF ((eIntegralConstantUnit = E_BA_Unit.eTime_Seconds OR eIntegralConstantUnit = 0) AND (eDerivativeConstantUnit = E_BA_Unit.eTime_Seconds)) AND
		((eDerivativeConstantUnit = E_BA_Unit.eTime_Seconds OR eDerivativeConstantUnit = 0) AND (eIntegralConstantUnit = E_BA_Unit.eTime_Seconds)) AND
		(ePropertionalConstantUnit = E_BA_Unit.eOther_NoUnits) THEN
		// Both are time_seconds:
		eMode := E_BACnet_LoopMode.eStandard;
		
	ELSIF (eIntegralConstantUnit <> E_BA_Unit.eTime_Seconds) AND
		(eDerivativeConstantUnit <> E_BA_Unit.eTime_Seconds) AND
		(ePropertionalConstantUnit = E_BA_Unit.eOther_NoUnits) THEN
		// Both are not time_seconds:
		eMode := E_BACnet_LoopMode.eIdeal;
		
	ELSE
		// Unknown settings - stop controller:
		eMode := E_BACnet_LoopMode.eNone;
	END_IF

	IF (NOT bEn) THEN
		fbIntCtrl.bReset := TRUE;
		
	ELSIF (eReliability <> E_BACnet_Reliability.eNoFaultDetected) OR (eMode = E_BACnet_LoopMode.eNone) THEN
		fbIntCtrl.bReset := TRUE;

	ELSIF stStateFlags.bOutOfService THEN
		fbIntCtrl.bReset := TRUE;

	// Decide the control action (direct or reverse):
	ELSIF (eAction = E_BA_Action.eDirect) THEN
		fbIntCtrl.bReset := FALSE;
		fbIntCtrl.fPresentValue := fCtrlVar;
		fbIntCtrl.fSetpoint := fSetpoint;

	ELSIF (eAction = E_BA_Action.eReverse) THEN
		fbIntCtrl.bReset := FALSE;
		fbIntCtrl.fPresentValue := fSetpoint;
		fbIntCtrl.fSetpoint := fCtrlVar;

	ELSE
		// Unknown action:
		fbIntCtrl.bReset := TRUE;
	END_IF

	// Set parameter depending on mode:
	CASE eMode OF
		E_BACnet_LoopMode.eIdeal:
			fbIntCtrl.fKp := fPropertionalConstant;
			fbIntCtrl.fKi := fIntegralConstant;
			fbIntCtrl.fKd := fDerivativeConstant;
			
		E_BACnet_LoopMode.eStandard:
			// Kp = Kp:
			fbIntCtrl.fKp := fPropertionalConstant;
			
			// Ki = Kp / Ti:
			IF (fIntegralConstant <> 0.0) THEN
				fbIntCtrl.fKi := (fPropertionalConstant / fIntegralConstant);
			ELSE
				fbIntCtrl.fKi := 0.0;
			END_IF
			
			// Kd = Kp * Td:
			fbIntCtrl.fKd := (fPropertionalConstant * fDerivativeConstant);
			
	END_CASE

	// Call PID control function block:
	fbIntCtrl(
		fCtrlCycleTime := _tCycleTime,
		fBias := fBias,
		fTp := -1.0,
		fMinOutput := fMinOutput,
		fMaxOutput := fMaxOutput,
		fY => fbAccLimit.X
	);
END_IF

// Limit present value:
fbAccLimit(X:=fbIntCtrl.fY, Amax:=fAccLimit, Tcycle:=_tCycleTime, Y=>fPresentValue);

// Calculate proportional band:
IF (fMaxOutput > 0.0) AND (fMinOutput >= 0.0) THEN
	fPropBand := ((fPresentValue - fMinOutput) / (fMaxOutput - fMinOutput)) * 100.0;
ELSIF (fMaxOutput <= 0.0) AND (fMinOutput < 0.0) THEN
	fPropBand := ((fPresentValue - fMaxOutput) / (fMaxOutput - fMinOutput)) * 100.0;
ELSIF (fPresentValue > 0.0) AND (fMaxOutput > 0.0) THEN
	fPropBand := (fPresentValue / fMaxOutput) * 100.0;
ELSIF (fPresentValue < 0.0) AND (fMinOutput < 0.0) THEN
	fPropBand := (fPresentValue / fMinOutput) * -100.0;
ELSE
	fPropBand := 0.0;
END_IF

SUPER^();

METHOD PROTECTED OnObjectStateChanged
SUPER^.OnObjectStateChanged();

CASE (tState) OF
	TCOM_STATE.TCOM_STATE_PREOP:
		// SyncHandler:
		RequestSyncHandlers(0, 18);
		
		// Properties:
		EnableProperty(E_BACnetPropIdentifier.PropManipulatedVariableReference, FALSE);
		EnableProperty(E_BACnetPropIdentifier.PropControlledVariableReference, FALSE);
		EnableProperty(E_BACnetPropIdentifier.PropSetpointReference, FALSE);
		EnableProperty(E_BACnetPropIdentifier.PropControlledVariableUnits, FALSE);
		EnableProperty(E_BACnetPropIdentifier.PropUpdateInterval, FALSE);
		
		EnableProperty(E_BACnetPropIdentifier.PropPriorityForWriting, FALSE);
		
		WriteProtectProperty(E_BACnetPropIdentifier.PropSetpoint, TRUE);
		WriteProtectProperty(E_BACnetPropIdentifier.PropControlledVariableValue, TRUE);
		
	TCOM_STATE.TCOM_STATE_SAFEOP:
		SyncProperty(E_BACnetPropIdentifier.PropPresentValue, SIZEOF(fPresentValue), ADR(fPresentValue), 0, eSync_ToSupplement, TRUE);
		SyncProperty(E_BACnetPropIdentifier.PropSetpoint, SIZEOF(fSetpoint), ADR(fSetpoint), 0, eSync_ToSupplement, TRUE);
		SyncProperty(E_BACnetPropIdentifier.PropControlledVariableValue, SIZEOF(fCtrlVar), ADR(fCtrlVar), 0, eSync_ToSupplement, TRUE);
	
	TCOM_STATE.TCOM_STATE_OP:
		SyncProperty(E_BACnetPropIdentifier.PropOutputUnits, SIZEOF(eOutputUnit), ADR(eOutputUnit), 0, eFullSync_InitPLC, FALSE);
		SyncProperty(E_BACnetPropIdentifier.PropOutOfService, SIZEOF(bEnOutOfService), ADR(bEnOutOfService), 0, eFullSync_InitPLC, FALSE);
		SyncProperty(E_BACnetPropIdentifier.PropCovIncrement, SIZEOF(fCOVIncrement), ADR(fCOVIncrement), 0, eFullSync_InitPLC, FALSE);
		SyncProperty(E_BACnetPropIdentifier.PropProportionalConstant, SIZEOF(fPropertionalConstant), ADR(fPropertionalConstant), 0, eFullSync_InitPLC, FALSE);
		SyncProperty(E_BACnetPropIdentifier.PropProportionalConstantUnits, SIZEOF(ePropertionalConstantUnit), ADR(ePropertionalConstantUnit), 0, eFullSync_InitPLC, FALSE);
		SyncProperty(E_BACnetPropIdentifier.PropIntegralConstant, SIZEOF(fIntegralConstant), ADR(fIntegralConstant), 0, eFullSync_InitPLC, FALSE);
		SyncProperty(E_BACnetPropIdentifier.PropIntegralConstantUnits, SIZEOF(eIntegralConstantUnit), ADR(eIntegralConstantUnit), 0, eFullSync_InitPLC, FALSE);
		SyncProperty(E_BACnetPropIdentifier.PropDerivativeConstant, SIZEOF(fDerivativeConstant), ADR(fDerivativeConstant), 0, eFullSync_InitPLC, FALSE);
		SyncProperty(E_BACnetPropIdentifier.PropDerivativeConstantUnits, SIZEOF(eDerivativeConstantUnit), ADR(eDerivativeConstantUnit), 0, eFullSync_InitPLC, FALSE);
		SyncProperty(E_BACnetPropIdentifier.PropDeadband, SIZEOF(fDeadband), ADR(fDeadband), 0, eFullSync_InitPLC, FALSE);
		SyncProperty(E_BACnetPropIdentifier.PropErrorLimit, SIZEOF(fErrorLimit), ADR(fErrorLimit), 0, eFullSync_InitPLC, FALSE);
		SyncProperty(E_BACnetPropIdentifier.PropMinimumOutput, SIZEOF(fMinOutput), ADR(fMinOutput), 0, eFullSync_InitPLC, FALSE);
		SyncProperty(E_BACnetPropIdentifier.PropMaximumOutput, SIZEOF(fMaxOutput), ADR(fMaxOutput), 0, eFullSync_InitPLC, FALSE);
		SyncProperty(E_BACnetPropIdentifier.PropActionProp, SIZEOF(eAction), ADR(eAction), 0, eFullSync_InitPLC, FALSE);
		SyncProperty(E_BACnetPropIdentifier.PropBias, SIZEOF(fBias), ADR(fBias), 0, eFullSync_InitPLC, FALSE);
		
END_CASE
END_METHOD

METHOD FB_init : BOOL
VAR_INPUT
	bInitRetains : BOOL; // if TRUE, the retain variables are initialized (warm start / cold start)
	bInCopyCode : BOOL;  // if TRUE, the instance afterwards gets moved into the copy code (online change)
END_VAR
eObjectType := E_BACnetObjType.ObjLoop;
END_METHOD

PROPERTY Mode : E_BACnet_LoopMode
GET
Mode := eMode;
END_GET
END_PROPERTY

PROPERTY ProportionalBand : REAL
GET
ProportionalBand := fPropBand;
END_GET
END_PROPERTY

END_FUNCTION_BLOCK

// POUs/Local/Objects/FB_BACnet_MI_IO
// Multistate Input Object
// - Terminal communication
FUNCTION_BLOCK FB_BACnet_MI_IO EXTENDS FB_BACnet_BaseMI
VAR_INPUT CONSTANT PERSISTENT
	{region 'Variable Parameters'}
		{attribute 'parameterCategory':='Config'}
		eMappingMode : E_BA_ByteMappingMode := E_BA_ByteMappingMode.eIndex1N;
		
		// Used value when no raw-value is active.
		// Note: The mapped process value is shifted '+1' when it is higher than this default value.
		//       > In fact the default value sorts into the range of valid process values.
		{attribute 'parameterCategory':='Value'}
		nRelinquishDefault : UDINT := 1;
	{endregion}
END_VAR
VAR
	{region 'Raw I/O'}
		bRawValue		AT %I*	: ST_BA_Byte;				// Bus terminal value
	{endregion}
	{region 'Internal'}
		bLastRawValue			: BYTE;
	{endregion}
END_VAR
VAR_STAT
	// (BETA) ... Following symbols should be made non-static / thread safe!
	{region 'Temporary'}
		{attribute 'hide'}
		_bRawValue				: POINTER TO BYTE;
	{endregion}
END_VAR

_bRawValue := ADR(bRawValue);

IF bReady THEN	
	// Trigger change of value:
	IF (_bRawValue^ <> bLastRawValue) THEN
		bLastRawValue := _bRawValue^;
		F_BA_MapUDIFromRawByte(bRawValue, nPresentValue, eMappingMode, nRelinquishDefault);
	END_IF
ELSE
	// Set last value to a different value compared to actual raw value (So a COV is triggered when current instance becomes ready):
	bLastRawValue := (_bRawValue^+1);
	
	nPresentValue := nRelinquishDefault;
END_IF

SUPER^();

END_FUNCTION_BLOCK

// POUs/Local/Objects/FB_BACnet_MI_Raw
// Multistate Input Object
// - Raw communication
FUNCTION_BLOCK FB_BACnet_MI_Raw EXTENDS FB_BACnet_BaseMI
VAR_INPUT
	nRawValue					: UDINT;			// Raw value
END_VAR

IF bReady THEN
	nPresentValue := nRawValue;
ELSE
	nPresentValue := 1;
END_IF

SUPER^();

END_FUNCTION_BLOCK

// POUs/Local/Objects/FB_BACnet_MV_Disp
// Multistate Setpoint Object for Setpoint
// - Used to display a value
FUNCTION_BLOCK FB_BACnet_MV_Disp EXTENDS FB_BACnet_Object
VAR_INPUT
	nVal				: UDINT		:= 1;
END_VAR
VAR_INPUT CONSTANT PERSISTENT
	{region 'Fixed Parameters'}
		{attribute 'parameterCategory':='Value'}
		{attribute 'TcEncoding':='UTF-8'}
		sStateText : ARRAY[1..BACnet_Param.nMultistate_StateCount] OF T_BACnet_StateText;
	{endregion}
END_VAR
VAR_OUTPUT
	nPresentValue		: UDINT		:= 1;
END_VAR
VAR
	{region 'Output-Properties'}
		nStateCount		: UDINT;
	{endregion}
END_VAR

IF bReady THEN
	nPresentValue := nVal;
ELSE
	nPresentValue := 1;
END_IF

SUPER^();

METHOD PROTECTED OnObjectStateChanged
SUPER^.OnObjectStateChanged();

CASE (tState) OF
	TCOM_STATE.TCOM_STATE_PREOP:
		// SyncHandler:
		{warning disable C0196}
		nStateCount := F_BACnet_GetUsedStateText(sStateText);
		{warning restore C0196}
		
		RequestSyncHandlers(0, nStateCount);								// Handlers for "E_BACnetPropIdentifier.PropStateText"
		RequestSyncHandlers(0, 1);											// Handlers for other properties
		
		// Properties:
		WriteProtectProperty(E_BACnetPropIdentifier.PropPresentValue, TRUE);
		WriteProtectProperty(E_BACnetPropIdentifier.PropNumberOfStates, TRUE);
		
		IF (BACnet_Param.bStateText_WriteProtect) THEN
			WriteProtectProperty(E_BACnetPropIdentifier.PropStateText, TRUE);
		END_IF
		
		EnableProperty(E_BACnetPropIdentifier.PropDeviceType, FALSE);
		EnableProperty(E_BACnetPropIdentifier.PropNotificationClass, FALSE);
		EnableProperty(E_BACnetPropIdentifier.PropNotifyType, FALSE);
		EnableProperty(E_BACnetPropIdentifier.PropEventEnable, FALSE);
		EnableProperty(E_BACnetPropIdentifier.PropEventTimeStamps, FALSE);
		EnableProperty(E_BACnetPropIdentifier.PropEventMessageTexts, FALSE);
		EnableProperty(E_BACnetPropIdentifier.PropEventMessageTextsConfig, FALSE);
		EnableProperty(E_BACnetPropIdentifier.PropTimeDelay, FALSE);
		EnableProperty(E_BACnetPropIdentifier.PropStatusFlags, FALSE);
		EnableProperty(E_BACnetPropIdentifier.PropAckedTransitions, FALSE);
		EnableProperty(E_BACnetPropIdentifier.PropReliability, FALSE);
		EnableProperty(E_BACnetPropIdentifier.PropEventState, FALSE);
		EnableProperty(E_BACnetPropIdentifier.PropEventDetectionEnable, FALSE);
		EnableProperty(E_BACnetPropIdentifier.PropEventAlgorithmInhibit, FALSE);
		EnableProperty(E_BACnetPropIdentifier.PropTimeDelayNormal, FALSE);
		EnableProperty(E_BACnetPropIdentifier.PropReliabilityEvaluationInhibit, FALSE);
		EnableProperty(E_BACnetPropIdentifier.PropAlarmValues, FALSE);
		EnableProperty(E_BACnetPropIdentifier.PropFaultValues, FALSE);
		EnableProperty(E_BACnetPropIdentifier.PropRelinquishDefault, FALSE);
		EnableProperty(E_BACnetPropIdentifier.PropPriorityArray, FALSE);
		EnableProperty(E_BACnetPropIdentifier.PropOutOfService, FALSE);
		EnableProperty(E_BACnetPropIdentifier.PropCurrentlyActivePriority, FALSE);
		
		// Ensure UTF-8 Encoding:
		F_BA_EnsureUTF8Array(ADR(sStateText), SIZEOF(sStateText[1]), TO_DINT(BACnet_Param.nMultistate_StateCount));
		
	TCOM_STATE.TCOM_STATE_SAFEOP:
		SyncProperty(E_BACnetPropIdentifier.PropPresentValue, SIZEOF(nVal), ADR(nVal), 0, eSync_ToSupplement, TRUE);
		
	TCOM_STATE.TCOM_STATE_OP:
		// Init number of used states:
		SetNumberOfStates(nStateCount);
		
		SyncPropertyList(E_BACnetPropIdentifier.PropStateText, ADR(sStateText), SIZEOF(T_BACnet_StateText), nStateCount, eFullSync_InitPLC, FALSE);

END_CASE
END_METHOD

METHOD FB_init : BOOL
VAR_INPUT
	bInitRetains : BOOL; // if TRUE, the retain variables are initialized (warm start / cold start)
	bInCopyCode : BOOL;  // if TRUE, the instance afterwards gets moved into the copy code (online change)
END_VAR
eObjectType := E_BACnetObjType.ObjMultistateValue;
END_METHOD

PROPERTY StateCount : UDINT
GET
StateCount := nStateCount;
END_GET
END_PROPERTY

END_FUNCTION_BLOCK

// POUs/Local/Objects/FB_BACnet_MV_Setp
// Multistate Setpoint Object for Setpoint
// - Used to define a setpoint by user
FUNCTION_BLOCK FB_BACnet_MV_Setp EXTENDS FB_BACnet_Object
VAR_INPUT CONSTANT PERSISTENT
	{region 'Fixed Parameters'}
		{attribute 'parameterCategory':='Value'}
		{attribute 'TcEncoding':='UTF-8'}
		sStateText : ARRAY[1..BACnet_Param.nMultistate_StateCount] OF T_BACnet_StateText;
	{endregion}
	{region 'Operational Parameters'}
		{attribute 'parameterCategory':='Value'}
		nValue : UDINT := 1;
	{endregion}
END_VAR
VAR_OUTPUT
	nPresentValue		: UDINT		:= 1;
END_VAR
VAR
	{region 'Output-Properties'}
		nStateCount		: UDINT;
	{endregion}
END_VAR

IF bReady THEN
	nPresentValue := nValue;
ELSE
	nPresentValue := 1;
END_IF

SUPER^();

METHOD PROTECTED OnObjectStateChanged
SUPER^.OnObjectStateChanged();

CASE (tState) OF
	TCOM_STATE.TCOM_STATE_PREOP:
		// SyncHandler:
		{warning disable C0196}
		nStateCount := F_BACnet_GetUsedStateText(sStateText);
		{warning restore C0196}
		
		RequestSyncHandlers(0, nStateCount);								// Handlers for "E_BACnetPropIdentifier.PropStateText"
		RequestSyncHandlers(0, 1);											// Handlers for other properties
		
		// Properties:
		WriteProtectProperty(E_BACnetPropIdentifier.PropNumberOfStates, TRUE);
		
		IF (BACnet_Param.bStateText_WriteProtect) THEN
			WriteProtectProperty(E_BACnetPropIdentifier.PropStateText, TRUE);
		END_IF
		
		EnableProperty(E_BACnetPropIdentifier.PropDeviceType, FALSE);
		EnableProperty(E_BACnetPropIdentifier.PropNotificationClass, FALSE);
		EnableProperty(E_BACnetPropIdentifier.PropNotifyType, FALSE);
		EnableProperty(E_BACnetPropIdentifier.PropEventEnable, FALSE);
		EnableProperty(E_BACnetPropIdentifier.PropEventTimeStamps, FALSE);
		EnableProperty(E_BACnetPropIdentifier.PropEventMessageTexts, FALSE);
		EnableProperty(E_BACnetPropIdentifier.PropEventMessageTextsConfig, FALSE);
		EnableProperty(E_BACnetPropIdentifier.PropTimeDelay, FALSE);
		EnableProperty(E_BACnetPropIdentifier.PropStatusFlags, FALSE);
		EnableProperty(E_BACnetPropIdentifier.PropAckedTransitions, FALSE);
		EnableProperty(E_BACnetPropIdentifier.PropReliability, FALSE);
		EnableProperty(E_BACnetPropIdentifier.PropEventState, FALSE);
		EnableProperty(E_BACnetPropIdentifier.PropEventDetectionEnable, FALSE);
		EnableProperty(E_BACnetPropIdentifier.PropEventAlgorithmInhibit, FALSE);
		EnableProperty(E_BACnetPropIdentifier.PropTimeDelayNormal, FALSE);
		EnableProperty(E_BACnetPropIdentifier.PropReliabilityEvaluationInhibit, FALSE);
		EnableProperty(E_BACnetPropIdentifier.PropAlarmValues, FALSE);
		EnableProperty(E_BACnetPropIdentifier.PropFaultValues, FALSE);
		EnableProperty(E_BACnetPropIdentifier.PropRelinquishDefault, FALSE);
		EnableProperty(E_BACnetPropIdentifier.PropPriorityArray, FALSE);
		EnableProperty(E_BACnetPropIdentifier.PropOutOfService, FALSE);
		EnableProperty(E_BACnetPropIdentifier.PropCurrentlyActivePriority, FALSE);
		
		// Ensure UTF-8 Encoding:
		F_BA_EnsureUTF8Array(ADR(sStateText), SIZEOF(sStateText[1]), TO_DINT(BACnet_Param.nMultistate_StateCount));
		
	TCOM_STATE.TCOM_STATE_SAFEOP:
		;
		
	TCOM_STATE.TCOM_STATE_OP:
		// Init number of used states:
		SetNumberOfStates(nStateCount);
		
		SyncProperty(E_BACnetPropIdentifier.PropPresentValue, SIZEOF(nValue), ADR(nValue), 0, eFullSync_InitPLC, FALSE);
		
		SyncPropertyList(E_BACnetPropIdentifier.PropStateText, ADR(sStateText), SIZEOF(T_BACnet_StateText), nStateCount, eFullSync_InitPLC, FALSE);

END_CASE
END_METHOD

METHOD FB_init : BOOL
VAR_INPUT
	bInitRetains : BOOL; // if TRUE, the retain variables are initialized (warm start / cold start)
	bInCopyCode : BOOL;  // if TRUE, the instance afterwards gets moved into the copy code (online change)
END_VAR
eObjectType := E_BACnetObjType.ObjMultistateValue;
END_METHOD

PROPERTY StateCount : UDINT
GET
StateCount := nStateCount;
END_GET
END_PROPERTY

END_FUNCTION_BLOCK

// POUs/Local/Objects/FB_BACnet_NC
// Notification Class Object
FUNCTION_BLOCK FB_BACnet_NC EXTENDS FB_BACnet_Object
VAR_INPUT CONSTANT PERSISTENT
	{region 'Variable Parameters'}
		{attribute 'parameterCategory':='Config'}
		nNotificationClass : UDINT;
		{attribute 'parameterCategory':='Config'}
		nPriority : ARRAY[E_BA_EventTransition.First .. E_BA_EventTransition.Last] OF UDINT;
		{attribute 'parameterCategory':='Config'}
		bAckRequired : ARRAY[E_BA_EventTransition.First .. E_BA_EventTransition.Last] OF BOOL;
		{attribute 'parameterCategory':='Config'}
		stRecipientList : ARRAY [1 .. BACnet_Param.nNC_RecipientArraySize] OF ST_BACnet_Destination;
	{endregion}
END_VAR
VAR_INPUT CONSTANT
	{region 'Variable Parameters'}
		{attribute 'parameterCategory':='Config'}
		bWriteRecipientList : BOOL;
	{endregion}
END_VAR
VAR
	{region 'COV'}
		bRecipientListChanged : BOOL;
	{endregion}
END_VAR

IF (bWriteRecipientList) THEN
	// (BETA) ... [DEBUG]
	F_BA_Print('Write RecipientList[1]', ADR(stRecipientList[1]), SIZEOF(stRecipientList[1]), TRUE, 64);
	
	bWriteRecipientList := FALSE;
	WritePropertyRecipientList(stRecipientList);
END_IF
IF (bRecipientListChanged) THEN
	bRecipientListChanged := FALSE;
	ReadPropertyRecipientList(stRecipientList);
	
	// (BETA) ... [DEBUG]
	F_BA_Print('Read RecipientList[1]', ADR(stRecipientList[1]), SIZEOF(stRecipientList[1]), TRUE, 64);
END_IF

SUPER^();

METHOD PROTECTED OnObjectStateChanged
SUPER^.OnObjectStateChanged();

CASE (tState) OF
	TCOM_STATE.TCOM_STATE_PREOP:
		// SyncHandler:
		RequestSyncHandlers(0, 7);
		
	TCOM_STATE.TCOM_STATE_SAFEOP:
		;
		
	TCOM_STATE.TCOM_STATE_OP:
		IF (SyncPropertyCOV(bRecipientListChanged, E_BACnetPropIdentifier.PropRecipientList)) THEN
			WritePropertyRecipientList(stRecipientList);
		END_IF
		
		SyncProperty(E_BACnetPropIdentifier.PropNotificationClass, SIZEOF(nNotificationClass), ADR(nNotificationClass), 0, eFullSync_InitPLC, FALSE);
		SyncPropertyIdx(E_BACnetPropIdentifier.PropPriority, SIZEOF(UDINT), ADR(nPriority[E_BA_EventTransition.eToOffnormal]), (E_BACnet_EventTransitionBits.eToOffnormal+1), 0, eFullSync_InitPLC, FALSE);	
		SyncPropertyIdx(E_BACnetPropIdentifier.PropPriority, SIZEOF(UDINT), ADR(nPriority[E_BA_EventTransition.eToFault]), (E_BACnet_EventTransitionBits.eToFault+1), 0, eFullSync_InitPLC, FALSE);	
		SyncPropertyIdx(E_BACnetPropIdentifier.PropPriority, SIZEOF(UDINT), ADR(nPriority[E_BA_EventTransition.eToNormal]), (E_BACnet_EventTransitionBits.eToNormal+1), 0, eFullSync_InitPLC, FALSE);
		SyncPropertyIdx(E_BACnetPropIdentifier.PropAckRequired, SIZEOF(BOOL), ADR(bAckRequired[E_BA_EventTransition.eToOffnormal]), E_BACnet_EventTransitionBits.eToOffnormal, 0, eFullSync_InitPLC, FALSE);	
		SyncPropertyIdx(E_BACnetPropIdentifier.PropAckRequired, SIZEOF(BOOL), ADR(bAckRequired[E_BA_EventTransition.eToFault]), E_BACnet_EventTransitionBits.eToFault, 0, eFullSync_InitPLC, FALSE);	
		SyncPropertyIdx(E_BACnetPropIdentifier.PropAckRequired, SIZEOF(BOOL), ADR(bAckRequired[E_BA_EventTransition.eToNormal]), E_BACnet_EventTransitionBits.eToNormal, 0, eFullSync_InitPLC, FALSE);
		
END_CASE
END_METHOD

METHOD FB_init : BOOL
VAR_INPUT
	bInitRetains : BOOL; // if TRUE, the retain variables are initialized (warm start / cold start)
	bInCopyCode : BOOL;  // if TRUE, the instance afterwards gets moved into the copy code (online change)
END_VAR
eObjectType := E_BACnetObjType.ObjNotificationClass;
END_METHOD

END_FUNCTION_BLOCK

// POUs/Local/Objects/FB_BACnet_PC
// Pulse Converter Object
FUNCTION_BLOCK FB_BACnet_PC EXTENDS FB_BACnet_EventObject
VAR_OUTPUT
	fPresentValue			: REAL;
END_VAR

SUPER^();

METHOD PROTECTED OnObjectStateChanged
SUPER^.OnObjectStateChanged();

CASE (tState) OF
	TCOM_STATE.TCOM_STATE_PREOP:
		// SyncHandler:
		RequestSyncHandlers(1, 0);
		
	TCOM_STATE.TCOM_STATE_SAFEOP:
		SyncProperty(E_BACnetPropIdentifier.PropPresentValue, SIZEOF(fPresentValue), ADR(fPresentValue), 0, eSync_FromSupplement, TRUE);
	
	TCOM_STATE.TCOM_STATE_OP:
		;
		
END_CASE
END_METHOD

METHOD FB_init : BOOL
VAR_INPUT
	bInitRetains : BOOL; // if TRUE, the retain variables are initialized (warm start / cold start)
	bInCopyCode : BOOL;  // if TRUE, the instance afterwards gets moved into the copy code (online change)
END_VAR
eObjectType := E_BACnetObjType.ObjPulseConverter;
END_METHOD

END_FUNCTION_BLOCK

// POUs/Local/Objects/FB_BACnet_Prog
// Program Object
FUNCTION_BLOCK FB_BACnet_Prog EXTENDS FB_BACnet_Object
VAR_OUTPUT
	eState			: E_BACnet_ProgramState;
END_VAR

SUPER^();

METHOD PROTECTED OnObjectStateChanged
SUPER^.OnObjectStateChanged();

CASE (tState) OF
	TCOM_STATE.TCOM_STATE_PREOP:
		// SyncHandler:
		RequestSyncHandlers(1, 0);
		
	TCOM_STATE.TCOM_STATE_SAFEOP:
		;
	
	TCOM_STATE.TCOM_STATE_OP:
		SyncProperty(E_BACnetPropIdentifier.PropProgramState, SIZEOF(eState), ADR(eState), 0, eSync_FromSupplement, FALSE);
		
END_CASE
END_METHOD

METHOD FB_init : BOOL
VAR_INPUT
	bInitRetains : BOOL; // if TRUE, the retain variables are initialized (warm start / cold start)
	bInCopyCode : BOOL;  // if TRUE, the instance afterwards gets moved into the copy code (online change)
END_VAR
eObjectType := E_BACnetObjType.ObjProg;
END_METHOD

END_FUNCTION_BLOCK

// POUs/Local/Objects/FB_BACnet_SchedA
// Analog Scheduler Object
FUNCTION_BLOCK FB_BACnet_SchedA EXTENDS FB_BACnet_BaseSched
VAR_INPUT CONSTANT PERSISTENT
	{region 'Fixed Parameters'}
		{attribute 'parameterCategory':='Value'}
		fScheduleDefault : REAL;
	{endregion}
END_VAR
VAR_OUTPUT
	fPresentValue		: REAL;
END_VAR

SUPER^();

METHOD PROTECTED OnObjectStateChanged
SUPER^.OnObjectStateChanged();

CASE (tState) OF
	TCOM_STATE.TCOM_STATE_PREOP:
		// SyncHandler:
		RequestSyncHandlers(1, 6);
		
	TCOM_STATE.TCOM_STATE_SAFEOP:
		;
		
	TCOM_STATE.TCOM_STATE_OP:
		SyncProperty(E_BACnetPropIdentifier.PropPresentValueReal, SIZEOF(fPresentValue), ADR(fPresentValue), 0, eSync_FromSupplement, FALSE);
		
		WritePropertyValueEx(E_BACnetPropIdentifier.PropScheduleDefault, eDatatype, SIZEOF(fScheduleDefault), ADR(fScheduleDefault));
		
END_CASE
END_METHOD

METHOD FB_init : BOOL
VAR_INPUT
	bInitRetains : BOOL; // if TRUE, the retain variables are initialized (warm start / cold start)
	bInCopyCode : BOOL;  // if TRUE, the instance afterwards gets moved into the copy code (online change)
END_VAR
eDatatype := E_BACnet_ValueChoice.eRealValue;

// Init default values:
tWeek := F_BACnet_SchedWeekly1xA(E_BA_Weekday.eMonday, E_BA_Weekday.eFriday, T#0H, 0.0);
END_METHOD

END_FUNCTION_BLOCK

// POUs/Local/Objects/FB_BACnet_SchedB
// Binary Scheduler Object
FUNCTION_BLOCK FB_BACnet_SchedB EXTENDS FB_BACnet_BaseSched
VAR_INPUT
	{attribute 'parameterUnit':= 's'}
	nPredictTime : UDINT;
END_VAR
VAR_INPUT CONSTANT PERSISTENT
	{region 'Fixed Parameters'}
		{attribute 'parameterCategory':='Value'}
		bScheduleDefault 	: BOOL;
	{endregion}
END_VAR
VAR_OUTPUT
	bPresentValue			: BOOL;
	bPredictedValue			: BOOL;
END_VAR

SUPER^();

METHOD PROTECTED OnObjectStateChanged
VAR
	_ePropPresentVal		: E_BACnetPropIdentifier;
END_VAR
SUPER^.OnObjectStateChanged();

CASE (tState) OF
	TCOM_STATE.TCOM_STATE_PREOP:
		// SyncHandler:
		RequestSyncHandlers(2, 1);
		
	TCOM_STATE.TCOM_STATE_SAFEOP:
		;
		
	TCOM_STATE.TCOM_STATE_OP:
		CASE (eDatatype) OF
			E_BACnet_ValueChoice.eEnumerationValue:
				_ePropPresentVal := E_BACnetPropIdentifier.PropPresentValueEnumerated;
			E_BACnet_ValueChoice.eBoolValue:
				_ePropPresentVal := E_BACnetPropIdentifier.PropPresentValueBool;
		ELSE
			iOwner.LogMsg.Show1(ADSLOG_MSGTYPE_ERROR, 'OOSC17', 'Property-synchronization aborted: Invalid datatype "%d"!', F_INT(eDatatype), FALSE);		
			RETURN;
		END_CASE

		SyncProperty(_ePropPresentVal, SIZEOF(bPresentValue), ADR(bPresentValue), 0, eSync_FromSupplement, FALSE);
		SyncProperty(E_BACnetPropIdentifier.PropPredictedScheduleBoolValue, SIZEOF(bPredictedValue), ADR(bPredictedValue), 0, eSync_FromSupplement, FALSE);

		SyncProperty(E_BACnetPropIdentifier.PropPredictScheduleValueTime, SIZEOF(nPredictTime), ADR(nPredictTime), 0, eSync_ToSupplement, FALSE);

		WritePropertyValueEx(E_BACnetPropIdentifier.PropScheduleDefault, eDatatype, SIZEOF(bScheduleDefault), ADR(bScheduleDefault));
		
END_CASE
END_METHOD

METHOD FB_init : BOOL
VAR_INPUT
	bInitRetains : BOOL; // if TRUE, the retain variables are initialized (warm start / cold start)
	bInCopyCode : BOOL;  // if TRUE, the instance afterwards gets moved into the copy code (online change)
END_VAR
CASE (BACnet_Param.eSched_BType) OF
	E_BACnet_SchedBType.eBinaryPV:
		eDatatype := E_BACnet_ValueChoice.eEnumerationValue;
	E_BACnet_SchedBType.eBool:
		eDatatype := E_BACnet_ValueChoice.eBoolValue;
END_CASE

// Init default values:
tWeek := F_BACnet_SchedWeekly1xB(E_BA_Weekday.eMonday, E_BA_Weekday.eFriday, T#0H, FALSE);
END_METHOD

END_FUNCTION_BLOCK

// POUs/Local/Objects/FB_BACnet_SchedM
// Multistate Scheduler Object
FUNCTION_BLOCK FB_BACnet_SchedM EXTENDS FB_BACnet_BaseSched
VAR_INPUT CONSTANT PERSISTENT
	{region 'Fixed Parameters'}
		{attribute 'parameterCategory':='Value'}
		nScheduleDefault : UDINT;
	{endregion}
END_VAR
VAR_OUTPUT
	nPresentValue		: UDINT;
END_VAR

SUPER^();

METHOD PROTECTED OnObjectStateChanged
SUPER^.OnObjectStateChanged();

CASE (tState) OF
	TCOM_STATE.TCOM_STATE_PREOP:
		// SyncHandler:
		RequestSyncHandlers(1, 0);
		
	TCOM_STATE.TCOM_STATE_SAFEOP:
		;
		
	TCOM_STATE.TCOM_STATE_OP:
		SyncProperty(E_BACnetPropIdentifier.PropPresentValueUnsigned, SIZEOF(nPresentValue), ADR(nPresentValue), 0, eSync_FromSupplement, FALSE);
		
		WritePropertyValueEx(E_BACnetPropIdentifier.PropScheduleDefault, eDatatype, SIZEOF(nScheduleDefault), ADR(nScheduleDefault));
		
END_CASE
END_METHOD

METHOD FB_init : BOOL
VAR_INPUT
	bInitRetains : BOOL; // if TRUE, the retain variables are initialized (warm start / cold start)
	bInCopyCode : BOOL;  // if TRUE, the instance afterwards gets moved into the copy code (online change)
END_VAR
eDatatype := E_BACnet_ValueChoice.eUnsignedValue;

// Init default values:
tWeek := F_BACnet_SchedWeekly1xM(E_BA_Weekday.eMonday, E_BA_Weekday.eFriday, T#0H, 1);
END_METHOD

END_FUNCTION_BLOCK

// POUs/Local/Objects/FB_BACnet_TLM



// (BETA) ... Implement FB
{attribute 'hide'}



FUNCTION_BLOCK FB_BACnet_TLM EXTENDS FB_BACnet_BaseTLog
VAR_INPUT CONSTANT PERSISTENT
	{region 'Fixed Parameters'}
		// (BETA) ... Implement "LogBuffer(Multiple)"-Property
		//{attribute 'hide'}
		//{attribute 'parameterCategory':='Value'}
		//tLogBuffer : ARRAY [1 .. BACnet_Param.nTLM_ArraySize] OF ST_BACnet_TLMEntry;
	{endregion}
END_VAR
VAR PERSISTENT
	{region 'SubInit'}
		// (BETA) ... Implement "DeviceObjPropRef(Multiple)"-Property
		// ...
	{endregion}
END_VAR
VAR
	{region 'Buffers'}
		{attribute 'hide'}
		fbLogBuffer					: FB_BACnet_TLMBuffer			:= (iRefObject := THIS^);
	{endregion}
END_VAR

// Synchronize Buffers:
fbLogBuffer();

SUPER^();

METHOD PROTECTED OnObjectStateChanged
SUPER^.OnObjectStateChanged();

// Synchronize:
fbLogBuffer.OnObjectStateChanged(tState);

CASE (tState) OF
	TCOM_STATE.TCOM_STATE_PREOP:
		;
	
	TCOM_STATE.TCOM_STATE_SAFEOP:
		;

	TCOM_STATE.TCOM_STATE_OP:
		;
		
END_CASE
END_METHOD

METHOD FB_init : BOOL
VAR_INPUT
	bInitRetains : BOOL; // if TRUE, the retain variables are initialized (warm start / cold start)
	bInCopyCode : BOOL;  // if TRUE, the instance afterwards gets moved into the copy code (online change)
END_VAR
eObjectType := E_BACnetObjType.ObjTrendLogMultiple;
END_METHOD

END_FUNCTION_BLOCK

// POUs/Local/Objects/FB_BACnet_TLog



// (BETA) ... Implement FB
{attribute 'hide'}



FUNCTION_BLOCK FB_BACnet_TLog EXTENDS FB_BACnet_BaseTLog

// (BETA) ... Implement "LogBuffer"-Property
///////////////////////////////////////////////////////////////
VAR_INPUT CONSTANT
	bTrendLog_Write	: BOOL;
END_VAR
///////////////////////////////////////////////////////////////


VAR_INPUT CONSTANT PERSISTENT
	{region 'Variable Parameters'}
		{attribute 'parameterCategory':='Value'}
		tLogBuffer : T_BACnet_TLogBuffer;
			 
		{attribute 'parameterCategory':='Config'}
		stDeviceObjPropRef : ST_BACnet_ObjectPropertyReference;
	{endregion}
END_VAR
VAR
	{region 'Buffers'}
		{attribute 'hide'}
		fbLogBuffer					: FB_BACnet_TrendLogBuffer			:= (iRefObject := THIS^);
	{endregion}
	{region 'Internal'}
		bLogBufferChanged			: BOOL;
	{endregion}
END_VAR

// Synchronize Buffers:
fbLogBuffer();

// (BETA) ... Implement "LogBuffer"-Property
///////////////////////////////////////////////////////////////
IF bTrendLog_Write THEN
	bTrendLog_Write := FALSE;
	{warning disable C0196}
	WritePropertyLogBuffer(tLogBuffer);
	{warning restore C0196}
END_IF
///////////////////////////////////////////////////////////////

IF bLogBufferChanged THEN
	bLogBufferChanged := FALSE;
	{warning disable C0196}
	ReadPropertyLogBuffer(tLogBuffer);
	{warning restore C0196}
END_IF

SUPER^();

METHOD PROTECTED OnObjectStateChanged
SUPER^.OnObjectStateChanged();

// Synchronize:
fbLogBuffer.OnObjectStateChanged(tState);

CASE (tState) OF
	TCOM_STATE.TCOM_STATE_PREOP:
		;
	
	TCOM_STATE.TCOM_STATE_SAFEOP:
		;

	TCOM_STATE.TCOM_STATE_OP:
		// Validate referred property:
		ValidateReference(stDeviceObjPropRef.iObject, stDeviceObjPropRef.tObjectID, 16#FF);
		
		// Initialize:
		IF (stDeviceObjPropRef.iObject <> 0) THEN
			// Initialize property reference:
			IF NOT stDeviceObjPropRef.iObject.Ready THEN
				// Initialize referred object bevor set reference in current instance:
				__QUERYPOINTER(stDeviceObjPropRef.iObject, _fbObjectTmp);
				_fbObjectTmp^();
			END_IF
				
			DeviceObjectPropertyReference := stDeviceObjPropRef;
		END_IF
		
END_CASE
END_METHOD

METHOD FB_init : BOOL
VAR_INPUT
	bInitRetains : BOOL; // if TRUE, the retain variables are initialized (warm start / cold start)
	bInCopyCode : BOOL;  // if TRUE, the instance afterwards gets moved into the copy code (online change)
END_VAR
eObjectType := E_BACnetObjType.ObjTrendLog;
END_METHOD

PROPERTY DeviceObjectPropertyReference : ST_BACnet_ObjectPropertyReference
GET
DeviceObjectPropertyReference := stDeviceObjPropRef;
END_GET
SET
stDeviceObjPropRef := DeviceObjectPropertyReference;

WritePropertyReference(E_BACnetPropIdentifier.PropLogDeviceObjectProperty, stDeviceObjPropRef);
END_SET
END_PROPERTY

END_FUNCTION_BLOCK

// POUs/Remote/Objects/Basic/[Base]/Basic/FB_BACnetRM_Object
FUNCTION_BLOCK FB_BACnetRM_Object EXTENDS FB_BACnetRM_BaseObject IMPLEMENTS I_BACnetRM_Object, I_BACnetRM_ObjectOwner
VAR
	{region 'Internal'}
		{attribute 'hide'}
		bParentInit					: BOOL := TRUE;
		{attribute 'hide'}
		fbLogMsg					: FB_BA_LogMessage;
	{endregion}
END_VAR

SUPER^();

// Unused - Implemented for compatibility reason!
{attribute 'hide'}
METHOD OnBACnetRMObjectCOV
VAR_INPUT
	ePropID		: E_BACnetPropIdentifier;
END_VAR
END_METHOD

// Unused - Implemented for compatibility reason!
{attribute 'hide'}
METHOD OnBACnetRMObjectStateChanged
END_METHOD

METHOD FB_init : BOOL
VAR_INPUT
	bInitRetains : BOOL; // if TRUE, the retain variables are initialized (warm start / cold start)
	bInCopyCode : BOOL;  // if TRUE, the instance afterwards gets moved into the copy code (online change)
END_VAR
iOwner := THIS^;
END_METHOD

{attribute 'suppress_wrn_C0410'}
{attribute 'hide'}
PROPERTY LogMsg : REFERENCE TO FB_BA_LogMessage
GET
LogMsg REF= fbLogMsg;
END_GET
END_PROPERTY

END_FUNCTION_BLOCK

